  [266] = {x=-22.822, y=-115.715, z=4.852, rx=175.392, ry=-0.809, rz=115, fatherId=fPrdFrame[0]}
  [267] = {x=-24.305, y=-115.715, z=4.874, rx=175.392, ry=-0.869, rz=115, fatherId=fPrdFrame[0]}
  [268] = {x=-25.789, y=-115.715, z=4.897, rx=175.392, ry=-0.928, rz=115, fatherId=fPrdFrame[0]}
  [269] = {x=-27.272, y=-115.714, z=4.922, rx=175.392, ry=-0.987, rz=115, fatherId=fPrdFrame[0]}
  [270] = {x=-28.756, y=-115.714, z=4.949, rx=175.392, ry=-1.046, rz=115, fatherId=fPrdFrame[0]}
  [271] = {x=-30.239, y=-115.714, z=4.977, rx=175.391, ry=-1.105, rz=115, fatherId=fPrdFrame[0]}
  [272] = {x=-31.723, y=-115.714, z=5.007, rx=175.391, ry=-1.165, rz=115, fatherId=fPrdFrame[0]}
  [273] = {x=-33.206, y=-115.714, z=5.038, rx=175.391, ry=-1.224, rz=115, fatherId=fPrdFrame[0]}
  [274] = {x=-34.69, y=-115.714, z=5.071, rx=175.391, ry=-1.283, rz=115, fatherId=fPrdFrame[0]}
  [275] = {x=-36.173, y=-115.714, z=5.105, rx=175.391, ry=-1.342, rz=115, fatherId=fPrdFrame[0]}
  [276] = {x=-37.657, y=-115.714, z=5.141, rx=175.391, ry=-1.401, rz=115, fatherId=fPrdFrame[0]}
  [277] = {x=-39.14, y=-115.714, z=5.179, rx=175.391, ry=-1.461, rz=115, fatherId=fPrdFrame[0]}
  [278] = {x=-40.624, y=-115.714, z=5.218, rx=175.391, ry=-1.52, rz=115, fatherId=fPrdFrame[0]}
  [279] = {x=-42.107, y=-115.714, z=5.258, rx=175.391, ry=-1.579, rz=115, fatherId=fPrdFrame[0]}
  [280] = {x=-43.591, y=-115.714, z=5.301, rx=175.39, ry=-1.638, rz=115, fatherId=fPrdFrame[0]}
  [281] = {x=-45.074, y=-115.714, z=5.344, rx=175.39, ry=-1.698, rz=115, fatherId=fPrdFrame[0]}
  [282] = {x=-46.557, y=-115.714, z=5.389, rx=175.39, ry=-1.757, rz=115, fatherId=fPrdFrame[0]}
  [283] = {x=-48.041, y=-115.714, z=5.436, rx=175.39, ry=-1.816, rz=115, fatherId=fPrdFrame[0]}
  [284] = {x=-49.524, y=-115.714, z=5.485, rx=175.39, ry=-1.875, rz=115, fatherId=fPrdFrame[0]}
  [285] = {x=-52.491, y=-114.23, z=5.466, rx=175.449, ry=-1.994, rz=115, fatherId=fPrdFrame[0]}
  [286] = {x=-51.008, y=-114.23, z=5.414, rx=175.449, ry=-1.934, rz=115, fatherId=fPrdFrame[0]}
  [287] = {x=-49.524, y=-114.23, z=5.364, rx=175.449, ry=-1.875, rz=115, fatherId=fPrdFrame[0]}
  [288] = {x=-48.041, y=-114.231, z=5.316, rx=175.449, ry=-1.816, rz=115, fatherId=fPrdFrame[0]}
  [289] = {x=-46.558, y=-114.231, z=5.269, rx=175.449, ry=-1.757, rz=115, fatherId=fPrdFrame[0]}
  [290] = {x=-45.074, y=-114.231, z=5.224, rx=175.45, ry=-1.697, rz=115, fatherId=fPrdFrame[0]}
  [291] = {x=-43.591, y=-114.231, z=5.18, rx=175.45, ry=-1.638, rz=115, fatherId=fPrdFrame[0]}
  [292] = {x=-42.107, y=-114.231, z=5.138, rx=175.45, ry=-1.579, rz=115, fatherId=fPrdFrame[0]}
  [293] = {x=-40.624, y=-114.231, z=5.098, rx=175.45, ry=-1.52, rz=115, fatherId=fPrdFrame[0]}
  [294] = {x=-39.14, y=-114.231, z=5.059, rx=175.45, ry=-1.461, rz=115, fatherId=fPrdFrame[0]}
  [295] = {x=-37.657, y=-114.231, z=5.021, rx=175.45, ry=-1.401, rz=115, fatherId=fPrdFrame[0]}
  [296] = {x=-36.173, y=-114.231, z=4.985, rx=175.45, ry=-1.342, rz=115, fatherId=fPrdFrame[0]}
  [297] = {x=-34.69, y=-114.231, z=4.951, rx=175.45, ry=-1.283, rz=115, fatherId=fPrdFrame[0]}
  [298] = {x=-33.206, y=-114.231, z=4.918, rx=175.45, ry=-1.224, rz=115, fatherId=fPrdFrame[0]}
  [299] = {x=-31.723, y=-114.231, z=4.887, rx=175.451, ry=-1.164, rz=115, fatherId=fPrdFrame[0]}
  [300] = {x=-30.239, y=-114.231, z=4.857, rx=175.451, ry=-1.105, rz=115, fatherId=fPrdFrame[0]}
  [301] = {x=-28.756, y=-114.231, z=4.829, rx=175.451, ry=-1.046, rz=115, fatherId=fPrdFrame[0]}
  [302] = {x=-27.272, y=-114.231, z=4.802, rx=175.451, ry=-0.987, rz=115, fatherId=fPrdFrame[0]}
  [303] = {x=-25.789, y=-114.231, z=4.777, rx=175.451, ry=-0.928, rz=115, fatherId=fPrdFrame[0]}
  [304] = {x=-24.305, y=-114.231, z=4.754, rx=175.451, ry=-0.868, rz=115, fatherId=fPrdFrame[0]}
  [305] = {x=-22.822, y=-114.231, z=4.732, rx=175.451, ry=-0.809, rz=115, fatherId=fPrdFrame[0]}
  [306] = {x=-21.339, y=-114.231, z=4.711, rx=175.451, ry=-0.75, rz=115, fatherId=fPrdFrame[0]}
  [307] = {x=-19.855, y=-114.231, z=4.693, rx=175.451, ry=-0.691, rz=115, fatherId=fPrdFrame[0]}
  [308] = {x=-18.372, y=-114.231, z=4.675, rx=175.451, ry=-0.632, rz=115, fatherId=fPrdFrame[0]}
  [309] = {x=-16.888, y=-114.231, z=4.659, rx=175.451, ry=-0.572, rz=115, fatherId=fPrdFrame[0]}
  [310] = {x=-15.405, y=-114.231, z=4.645, rx=175.451, ry=-0.513, rz=115, fatherId=fPrdFrame[0]}
  [311] = {x=-13.921, y=-114.231, z=4.633, rx=175.451, ry=-0.454, rz=115, fatherId=fPrdFrame[0]}
  [312] = {x=-12.438, y=-114.231, z=4.621, rx=175.451, ry=-0.395, rz=115, fatherId=fPrdFrame[0]}
  [313] = {x=-10.954, y=-114.231, z=4.612, rx=175.451, ry=-0.336, rz=115, fatherId=fPrdFrame[0]}
  [314] = {x=-9.471, y=-114.231, z=4.604, rx=175.451, ry=-0.276, rz=115, fatherId=fPrdFrame[0]}
  [315] = {x=-7.987, y=-114.231, z=4.597, rx=175.451, ry=-0.217, rz=115, fatherId=fPrdFrame[0]}
  [316] = {x=-6.504, y=-114.231, z=4.592, rx=175.451, ry=-0.158, rz=115, fatherId=fPrdFrame[0]}
  [317] = {x=-5.02, y=-114.231, z=4.589, rx=175.451, ry=-0.099, rz=115, fatherId=fPrdFrame[0]}
  [318] = {x=-3.537, y=-114.231, z=4.587, rx=175.451, ry=-0.04, rz=115, fatherId=fPrdFrame[0]}
  [319] = {x=-2.053, y=-114.231, z=4.587, rx=175.451, ry=0.02, rz=115, fatherId=fPrdFrame[0]}
  [320] = {x=-0.57, y=-114.231, z=4.588, rx=175.451, ry=0.079, rz=115, fatherId=fPrdFrame[0]}
  [321] = {x=0.913, y=-114.231, z=4.591, rx=175.451, ry=0.138, rz=115, fatherId=fPrdFrame[0]}
  [322] = {x=2.397, y=-114.231, z=4.596, rx=175.451, ry=0.197, rz=115, fatherId=fPrdFrame[0]}
  [323] = {x=3.88, y=-114.231, z=4.601, rx=175.451, ry=0.256, rz=115, fatherId=fPrdFrame[0]}
  [324] = {x=5.364, y=-114.231, z=4.609, rx=175.451, ry=0.316, rz=115, fatherId=fPrdFrame[0]}
  [325] = {x=6.847, y=-114.231, z=4.618, rx=175.451, ry=0.375, rz=115, fatherId=fPrdFrame[0]}
  [326] = {x=8.331, y=-114.231, z=4.629, rx=175.451, ry=0.434, rz=115, fatherId=fPrdFrame[0]}
  [327] = {x=9.814, y=-114.231, z=4.641, rx=175.451, ry=0.493, rz=115, fatherId=fPrdFrame[0]}
  [328] = {x=11.298, y=-114.231, z=4.654, rx=175.451, ry=0.552, rz=115, fatherId=fPrdFrame[0]}
  [329] = {x=12.781, y=-114.231, z=4.67, rx=175.451, ry=0.612, rz=115, fatherId=fPrdFrame[0]}
  [330] = {x=14.265, y=-114.231, z=4.686, rx=175.451, ry=0.671, rz=115, fatherId=fPrdFrame[0]}
  [331] = {x=15.748, y=-114.231, z=4.705, rx=175.451, ry=0.73, rz=115, fatherId=fPrdFrame[0]}
  [332] = {x=17.232, y=-114.231, z=4.725, rx=175.451, ry=0.789, rz=115, fatherId=fPrdFrame[0]}
  [333] = {x=18.715, y=-114.231, z=4.746, rx=175.451, ry=0.848, rz=115, fatherId=fPrdFrame[0]}
  [334] = {x=20.199, y=-114.231, z=4.769, rx=175.451, ry=0.908, rz=115, fatherId=fPrdFrame[0]}
  [335] = {x=21.682, y=-114.231, z=4.794, rx=175.451, ry=0.967, rz=115, fatherId=fPrdFrame[0]}
  [336] = {x=23.166, y=-114.231, z=4.82, rx=175.451, ry=1.026, rz=115, fatherId=fPrdFrame[0]}
  [337] = {x=24.649, y=-114.231, z=4.847, rx=175.451, ry=1.085, rz=115, fatherId=fPrdFrame[0]}
  [338] = {x=26.132, y=-114.231, z=4.877, rx=175.451, ry=1.144, rz=115, fatherId=fPrdFrame[0]}
  [339] = {x=27.616, y=-114.231, z=4.907, rx=175.45, ry=1.204, rz=115, fatherId=fPrdFrame[0]}
  [340] = {x=29.099, y=-114.231, z=4.94, rx=175.45, ry=1.263, rz=115, fatherId=fPrdFrame[0]}
  [341] = {x=30.583, y=-114.231, z=4.973, rx=175.45, ry=1.322, rz=115, fatherId=fPrdFrame[0]}
  [342] = {x=32.066, y=-114.231, z=5.009, rx=175.45, ry=1.381, rz=115, fatherId=fPrdFrame[0]}
  [343] = {x=33.55, y=-114.231, z=5.046, rx=175.45, ry=1.44, rz=115, fatherId=fPrdFrame[0]}
  [344] = {x=35.033, y=-114.231, z=5.084, rx=175.45, ry=1.5, rz=115, fatherId=fPrdFrame[0]}
  [345] = {x=36.517, y=-114.231, z=5.124, rx=175.45, ry=1.559, rz=115, fatherId=fPrdFrame[0]}
  [346] = {x=38, y=-114.231, z=5.166, rx=175.45, ry=1.618, rz=115, fatherId=fPrdFrame[0]}
  [347] = {x=39.484, y=-114.231, z=5.209, rx=175.45, ry=1.677, rz=115, fatherId=fPrdFrame[0]}
  [348] = {x=40.967, y=-114.231, z=5.254, rx=175.449, ry=1.736, rz=115, fatherId=fPrdFrame[0]}
  [349] = {x=42.451, y=-114.231, z=5.3, rx=175.449, ry=1.796, rz=115, fatherId=fPrdFrame[0]}
  [350] = {x=43.934, y=-114.23, z=5.348, rx=175.449, ry=1.855, rz=115, fatherId=fPrdFrame[0]}
  [351] = {x=45.418, y=-114.23, z=5.397, rx=175.449, ry=1.914, rz=115, fatherId=fPrdFrame[0]}
  [352] = {x=46.901, y=-114.23, z=5.448, rx=175.449, ry=1.973, rz=115, fatherId=fPrdFrame[0]}
  [353] = {x=51.351, y=-112.747, z=5.491, rx=175.508, ry=2.151, rz=115, fatherId=fPrdFrame[0]}
  [354] = {x=49.868, y=-112.747, z=5.436, rx=175.508, ry=2.092, rz=115, fatherId=fPrdFrame[0]}
  [355] = {x=48.385, y=-112.747, z=5.382, rx=175.508, ry=2.032, rz=115, fatherId=fPrdFrame[0]}
  [356] = {x=46.901, y=-112.747, z=5.329, rx=175.508, ry=1.973, rz=115, fatherId=fPrdFrame[0]}
  [357] = {x=45.418, y=-112.747, z=5.278, rx=175.508, ry=1.914, rz=115, fatherId=fPrdFrame[0]}
  [358] = {x=43.934, y=-112.747, z=5.229, rx=175.508, ry=1.855, rz=115, fatherId=fPrdFrame[0]}
  [359] = {x=42.451, y=-112.747, z=5.181, rx=175.508, ry=1.796, rz=115, fatherId=fPrdFrame[0]}
  [360] = {x=40.967, y=-112.747, z=5.135, rx=175.509, ry=1.736, rz=115, fatherId=fPrdFrame[0]}
  [361] = {x=39.484, y=-112.747, z=5.09, rx=175.509, ry=1.677, rz=115, fatherId=fPrdFrame[0]}
  [362] = {x=38, y=-112.747, z=5.047, rx=175.509, ry=1.618, rz=115, fatherId=fPrdFrame[0]}
  [363] = {x=36.517, y=-112.747, z=5.006, rx=175.509, ry=1.559, rz=115, fatherId=fPrdFrame[0]}
  [364] = {x=35.033, y=-112.747, z=4.966, rx=175.509, ry=1.499, rz=115, fatherId=fPrdFrame[0]}
  [365] = {x=33.55, y=-112.747, z=4.927, rx=175.509, ry=1.44, rz=115, fatherId=fPrdFrame[0]}
  [366] = {x=32.066, y=-112.747, z=4.89, rx=175.509, ry=1.381, rz=115, fatherId=fPrdFrame[0]}
  [367] = {x=30.583, y=-112.747, z=4.855, rx=175.51, ry=1.322, rz=115, fatherId=fPrdFrame[0]}
  [368] = {x=29.099, y=-112.747, z=4.821, rx=175.51, ry=1.263, rz=115, fatherId=fPrdFrame[0]}
  [369] = {x=27.616, y=-112.747, z=4.789, rx=175.51, ry=1.203, rz=115, fatherId=fPrdFrame[0]}
  [370] = {x=26.132, y=-112.747, z=4.758, rx=175.51, ry=1.144, rz=115, fatherId=fPrdFrame[0]}
  [371] = {x=24.649, y=-112.747, z=4.729, rx=175.51, ry=1.085, rz=115, fatherId=fPrdFrame[0]}
  [372] = {x=23.166, y=-112.747, z=4.701, rx=175.51, ry=1.026, rz=115, fatherId=fPrdFrame[0]}
  [373] = {x=21.682, y=-112.747, z=4.675, rx=175.51, ry=0.967, rz=115, fatherId=fPrdFrame[0]}
  [374] = {x=20.199, y=-112.747, z=4.651, rx=175.51, ry=0.907, rz=115, fatherId=fPrdFrame[0]}
  [375] = {x=18.715, y=-112.747, z=4.628, rx=175.51, ry=0.848, rz=115, fatherId=fPrdFrame[0]}
  [376] = {x=17.232, y=-112.748, z=4.606, rx=175.51, ry=0.789, rz=115, fatherId=fPrdFrame[0]}
  [377] = {x=15.748, y=-112.748, z=4.586, rx=175.51, ry=0.73, rz=115, fatherId=fPrdFrame[0]}
  [378] = {x=14.265, y=-112.748, z=4.568, rx=175.51, ry=0.671, rz=115, fatherId=fPrdFrame[0]}
  [379] = {x=12.781, y=-112.748, z=4.551, rx=175.51, ry=0.611, rz=115, fatherId=fPrdFrame[0]}
  [380] = {x=11.298, y=-112.748, z=4.536, rx=175.51, ry=0.552, rz=115, fatherId=fPrdFrame[0]}
  [381] = {x=9.814, y=-112.748, z=4.522, rx=175.511, ry=0.493, rz=115, fatherId=fPrdFrame[0]}
  [382] = {x=8.331, y=-112.748, z=4.51, rx=175.511, ry=0.434, rz=115, fatherId=fPrdFrame[0]}
  [383] = {x=6.847, y=-112.748, z=4.499, rx=175.511, ry=0.375, rz=115, fatherId=fPrdFrame[0]}
  [384] = {x=5.364, y=-112.748, z=4.49, rx=175.511, ry=0.315, rz=115, fatherId=fPrdFrame[0]}
  [385] = {x=3.88, y=-112.748, z=4.483, rx=175.511, ry=0.256, rz=115, fatherId=fPrdFrame[0]}
  [386] = {x=2.397, y=-112.748, z=4.477, rx=175.511, ry=0.197, rz=115, fatherId=fPrdFrame[0]}
  [387] = {x=0.913, y=-112.748, z=4.473, rx=175.511, ry=0.138, rz=115, fatherId=fPrdFrame[0]}
  [388] = {x=-0.57, y=-112.748, z=4.47, rx=175.511, ry=0.079, rz=115, fatherId=fPrdFrame[0]}
  [389] = {x=-2.053, y=-112.748, z=4.469, rx=175.511, ry=0.02, rz=115, fatherId=fPrdFrame[0]}
  [390] = {x=-3.537, y=-112.748, z=4.469, rx=175.511, ry=-0.04, rz=115, fatherId=fPrdFrame[0]}
  [391] = {x=-5.02, y=-112.748, z=4.471, rx=175.511, ry=-0.099, rz=115, fatherId=fPrdFrame[0]}
  [392] = {x=-6.504, y=-112.748, z=4.474, rx=175.511, ry=-0.158, rz=115, fatherId=fPrdFrame[0]}
  [393] = {x=-7.987, y=-112.748, z=4.479, rx=175.511, ry=-0.217, rz=115, fatherId=fPrdFrame[0]}
  [394] = {x=-9.471, y=-112.748, z=4.485, rx=175.511, ry=-0.276, rz=115, fatherId=fPrdFrame[0]}
  [395] = {x=-10.954, y=-112.748, z=4.493, rx=175.511, ry=-0.336, rz=115, fatherId=fPrdFrame[0]}
  [396] = {x=-12.438, y=-112.748, z=4.503, rx=175.511, ry=-0.395, rz=115, fatherId=fPrdFrame[0]}
  [397] = {x=-13.921, y=-112.748, z=4.514, rx=175.511, ry=-0.454, rz=115, fatherId=fPrdFrame[0]}
  [398] = {x=-15.405, y=-112.748, z=4.527, rx=175.511, ry=-0.513, rz=115, fatherId=fPrdFrame[0]}
  [399] = {x=-16.888, y=-112.748, z=4.541, rx=175.51, ry=-0.572, rz=115, fatherId=fPrdFrame[0]}
  [400] = {x=-18.372, y=-112.748, z=4.557, rx=175.51, ry=-0.632, rz=115, fatherId=fPrdFrame[0]}
  [401] = {x=-19.855, y=-112.748, z=4.574, rx=175.51, ry=-0.691, rz=115, fatherId=fPrdFrame[0]}
  [402] = {x=-21.339, y=-112.748, z=4.593, rx=175.51, ry=-0.75, rz=115, fatherId=fPrdFrame[0]}
  [403] = {x=-22.822, y=-112.748, z=4.613, rx=175.51, ry=-0.809, rz=115, fatherId=fPrdFrame[0]}
  [404] = {x=-24.306, y=-112.747, z=4.635, rx=175.51, ry=-0.868, rz=115, fatherId=fPrdFrame[0]}
  [405] = {x=-25.789, y=-112.747, z=4.659, rx=175.51, ry=-0.928, rz=115, fatherId=fPrdFrame[0]}
  [406] = {x=-27.272, y=-112.747, z=4.684, rx=175.51, ry=-0.987, rz=115, fatherId=fPrdFrame[0]}
  [407] = {x=-28.756, y=-112.747, z=4.71, rx=175.51, ry=-1.046, rz=115, fatherId=fPrdFrame[0]}
  [408] = {x=-30.239, y=-112.747, z=4.739, rx=175.51, ry=-1.105, rz=115, fatherId=fPrdFrame[0]}
  [409] = {x=-31.723, y=-112.747, z=4.768, rx=175.51, ry=-1.164, rz=115, fatherId=fPrdFrame[0]}
  [410] = {x=-33.206, y=-112.747, z=4.799, rx=175.51, ry=-1.224, rz=115, fatherId=fPrdFrame[0]}
  [411] = {x=-34.69, y=-112.747, z=4.832, rx=175.51, ry=-1.283, rz=115, fatherId=fPrdFrame[0]}
  [412] = {x=-36.173, y=-112.747, z=4.867, rx=175.509, ry=-1.342, rz=115, fatherId=fPrdFrame[0]}
  [413] = {x=-37.657, y=-112.747, z=4.903, rx=175.509, ry=-1.401, rz=115, fatherId=fPrdFrame[0]}
  [414] = {x=-39.14, y=-112.747, z=4.94, rx=175.509, ry=-1.46, rz=115, fatherId=fPrdFrame[0]}
  [415] = {x=-40.624, y=-112.747, z=4.979, rx=175.509, ry=-1.52, rz=115, fatherId=fPrdFrame[0]}
  [416] = {x=-42.107, y=-112.747, z=5.02, rx=175.509, ry=-1.579, rz=115, fatherId=fPrdFrame[0]}
  [417] = {x=-43.591, y=-112.747, z=5.062, rx=175.509, ry=-1.638, rz=115, fatherId=fPrdFrame[0]}
  [418] = {x=-45.074, y=-112.747, z=5.105, rx=175.509, ry=-1.697, rz=115, fatherId=fPrdFrame[0]}
  [419] = {x=-46.558, y=-112.747, z=5.151, rx=175.509, ry=-1.756, rz=115, fatherId=fPrdFrame[0]}
  [420] = {x=-48.041, y=-112.747, z=5.197, rx=175.508, ry=-1.816, rz=115, fatherId=fPrdFrame[0]}
  [421] = {x=-49.525, y=-112.747, z=5.246, rx=175.508, ry=-1.875, rz=115, fatherId=fPrdFrame[0]}
  [422] = {x=-51.008, y=-112.747, z=5.296, rx=175.508, ry=-1.934, rz=115, fatherId=fPrdFrame[0]}
  [423] = {x=-52.491, y=-112.747, z=5.347, rx=175.508, ry=-1.993, rz=115, fatherId=fPrdFrame[0]}
  [424] = {x=-53.975, y=-112.747, z=5.4, rx=175.508, ry=-2.053, rz=115, fatherId=fPrdFrame[0]}
  [425] = {x=-55.458, y=-112.747, z=5.455, rx=175.508, ry=-2.112, rz=115, fatherId=fPrdFrame[0]}
  [426] = {x=-58.425, y=-111.263, z=5.451, rx=175.567, ry=-2.23, rz=115, fatherId=fPrdFrame[0]}
  [427] = {x=-56.942, y=-111.263, z=5.394, rx=175.567, ry=-2.171, rz=115, fatherId=fPrdFrame[0]}
  [428] = {x=-55.458, y=-111.263, z=5.338, rx=175.567, ry=-2.112, rz=115, fatherId=fPrdFrame[0]}
  [429] = {x=-53.975, y=-111.263, z=5.283, rx=175.567, ry=-2.052, rz=115, fatherId=fPrdFrame[0]}
  [430] = {x=-52.492, y=-111.263, z=5.23, rx=175.567, ry=-1.993, rz=115, fatherId=fPrdFrame[0]}
  [431] = {x=-51.008, y=-111.263, z=5.179, rx=175.567, ry=-1.934, rz=115, fatherId=fPrdFrame[0]}
  [432] = {x=-49.525, y=-111.263, z=5.129, rx=175.568, ry=-1.875, rz=115, fatherId=fPrdFrame[0]}
  [433] = {x=-48.041, y=-111.263, z=5.08, rx=175.568, ry=-1.816, rz=115, fatherId=fPrdFrame[0]}
  [434] = {x=-46.558, y=-111.264, z=5.034, rx=175.568, ry=-1.756, rz=115, fatherId=fPrdFrame[0]}
  [435] = {x=-45.074, y=-111.264, z=4.988, rx=175.568, ry=-1.697, rz=115, fatherId=fPrdFrame[0]}
  [436] = {x=-43.591, y=-111.264, z=4.945, rx=175.568, ry=-1.638, rz=115, fatherId=fPrdFrame[0]}
  [437] = {x=-42.107, y=-111.264, z=4.903, rx=175.568, ry=-1.579, rz=115, fatherId=fPrdFrame[0]}
  [438] = {x=-40.624, y=-111.264, z=4.862, rx=175.568, ry=-1.519, rz=115, fatherId=fPrdFrame[0]}
  [439] = {x=-39.14, y=-111.264, z=4.823, rx=175.568, ry=-1.46, rz=115, fatherId=fPrdFrame[0]}
  [440] = {x=-37.657, y=-111.264, z=4.786, rx=175.569, ry=-1.401, rz=115, fatherId=fPrdFrame[0]}
  [441] = {x=-36.173, y=-111.264, z=4.75, rx=175.569, ry=-1.342, rz=115, fatherId=fPrdFrame[0]}
  [442] = {x=-34.69, y=-111.264, z=4.715, rx=175.569, ry=-1.283, rz=115, fatherId=fPrdFrame[0]}
  [443] = {x=-33.206, y=-111.264, z=4.682, rx=175.569, ry=-1.223, rz=115, fatherId=fPrdFrame[0]}
  [444] = {x=-31.723, y=-111.264, z=4.651, rx=175.569, ry=-1.164, rz=115, fatherId=fPrdFrame[0]}
  [445] = {x=-30.239, y=-111.264, z=4.622, rx=175.569, ry=-1.105, rz=115, fatherId=fPrdFrame[0]}
  [446] = {x=-28.756, y=-111.264, z=4.593, rx=175.569, ry=-1.046, rz=115, fatherId=fPrdFrame[0]}
  [447] = {x=-27.272, y=-111.264, z=4.567, rx=175.569, ry=-0.987, rz=115, fatherId=fPrdFrame[0]}
  [448] = {x=-25.789, y=-111.264, z=4.542, rx=175.569, ry=-0.927, rz=115, fatherId=fPrdFrame[0]}
  [449] = {x=-24.306, y=-111.264, z=4.518, rx=175.569, ry=-0.868, rz=115, fatherId=fPrdFrame[0]}
  [450] = {x=-22.822, y=-111.264, z=4.496, rx=175.569, ry=-0.809, rz=115, fatherId=fPrdFrame[0]}
  [451] = {x=-21.339, y=-111.264, z=4.476, rx=175.57, ry=-0.75, rz=115, fatherId=fPrdFrame[0]}
  [452] = {x=-19.855, y=-111.264, z=4.457, rx=175.57, ry=-0.691, rz=115, fatherId=fPrdFrame[0]}
  [453] = {x=-18.372, y=-111.264, z=4.44, rx=175.57, ry=-0.632, rz=115, fatherId=fPrdFrame[0]}
  [454] = {x=-16.888, y=-111.264, z=4.424, rx=175.57, ry=-0.572, rz=115, fatherId=fPrdFrame[0]}
  [455] = {x=-15.405, y=-111.264, z=4.41, rx=175.57, ry=-0.513, rz=115, fatherId=fPrdFrame[0]}
  [456] = {x=-13.921, y=-111.264, z=4.397, rx=175.57, ry=-0.454, rz=115, fatherId=fPrdFrame[0]}
  [457] = {x=-12.438, y=-111.264, z=4.386, rx=175.57, ry=-0.395, rz=115, fatherId=fPrdFrame[0]}
  [458] = {x=-10.954, y=-111.264, z=4.376, rx=175.57, ry=-0.336, rz=115, fatherId=fPrdFrame[0]}
  [459] = {x=-9.471, y=-111.264, z=4.368, rx=175.57, ry=-0.276, rz=115, fatherId=fPrdFrame[0]}
  [460] = {x=-7.987, y=-111.264, z=4.362, rx=175.57, ry=-0.217, rz=115, fatherId=fPrdFrame[0]}
  [461] = {x=-6.504, y=-111.264, z=4.357, rx=175.57, ry=-0.158, rz=115, fatherId=fPrdFrame[0]}
  [462] = {x=-5.02, y=-111.264, z=4.354, rx=175.57, ry=-0.099, rz=115, fatherId=fPrdFrame[0]}
  [463] = {x=-3.537, y=-111.264, z=4.352, rx=175.57, ry=-0.04, rz=115, fatherId=fPrdFrame[0]}
  [464] = {x=-2.053, y=-111.264, z=4.352, rx=175.57, ry=0.02, rz=115, fatherId=fPrdFrame[0]}
  [465] = {x=-0.57, y=-111.264, z=4.353, rx=175.57, ry=0.079, rz=115, fatherId=fPrdFrame[0]}
  [466] = {x=0.913, y=-111.264, z=4.356, rx=175.57, ry=0.138, rz=115, fatherId=fPrdFrame[0]}
  [467] = {x=2.397, y=-111.264, z=4.36, rx=175.57, ry=0.197, rz=115, fatherId=fPrdFrame[0]}
  [468] = {x=3.88, y=-111.264, z=4.366, rx=175.57, ry=0.256, rz=115, fatherId=fPrdFrame[0]}
  [469] = {x=5.364, y=-111.264, z=4.373, rx=175.57, ry=0.315, rz=115, fatherId=fPrdFrame[0]}
  [470] = {x=6.847, y=-111.264, z=4.382, rx=175.57, ry=0.375, rz=115, fatherId=fPrdFrame[0]}
  [471] = {x=8.331, y=-111.264, z=4.393, rx=175.57, ry=0.434, rz=115, fatherId=fPrdFrame[0]}
  [472] = {x=9.814, y=-111.264, z=4.405, rx=175.57, ry=0.493, rz=115, fatherId=fPrdFrame[0]}
  [473] = {x=11.298, y=-111.264, z=4.419, rx=175.57, ry=0.552, rz=115, fatherId=fPrdFrame[0]}
  [474] = {x=12.781, y=-111.264, z=4.434, rx=175.57, ry=0.611, rz=115, fatherId=fPrdFrame[0]}
  [475] = {x=14.265, y=-111.264, z=4.451, rx=175.57, ry=0.671, rz=115, fatherId=fPrdFrame[0]}
  [476] = {x=15.748, y=-111.264, z=4.469, rx=175.57, ry=0.73, rz=115, fatherId=fPrdFrame[0]}
  [477] = {x=17.232, y=-111.264, z=4.489, rx=175.569, ry=0.789, rz=115, fatherId=fPrdFrame[0]}
  [478] = {x=18.715, y=-111.264, z=4.511, rx=175.569, ry=0.848, rz=115, fatherId=fPrdFrame[0]}
  [479] = {x=20.199, y=-111.264, z=4.534, rx=175.569, ry=0.907, rz=115, fatherId=fPrdFrame[0]}
  [480] = {x=21.682, y=-111.264, z=4.558, rx=175.569, ry=0.967, rz=115, fatherId=fPrdFrame[0]}
  [481] = {x=23.166, y=-111.264, z=4.584, rx=175.569, ry=1.026, rz=115, fatherId=fPrdFrame[0]}
  [482] = {x=24.649, y=-111.264, z=4.612, rx=175.569, ry=1.085, rz=115, fatherId=fPrdFrame[0]}
  [483] = {x=26.133, y=-111.264, z=4.641, rx=175.569, ry=1.144, rz=115, fatherId=fPrdFrame[0]}
  [484] = {x=27.616, y=-111.264, z=4.672, rx=175.569, ry=1.203, rz=115, fatherId=fPrdFrame[0]}
  [485] = {x=29.099, y=-111.264, z=4.704, rx=175.569, ry=1.263, rz=115, fatherId=fPrdFrame[0]}
  [486] = {x=30.583, y=-111.264, z=4.738, rx=175.569, ry=1.322, rz=115, fatherId=fPrdFrame[0]}
  [487] = {x=32.066, y=-111.264, z=4.773, rx=175.569, ry=1.381, rz=115, fatherId=fPrdFrame[0]}
  [488] = {x=33.55, y=-111.264, z=4.81, rx=175.568, ry=1.44, rz=115, fatherId=fPrdFrame[0]}
  [489] = {x=35.033, y=-111.264, z=4.849, rx=175.568, ry=1.499, rz=115, fatherId=fPrdFrame[0]}
  [490] = {x=36.517, y=-111.264, z=4.889, rx=175.568, ry=1.559, rz=115, fatherId=fPrdFrame[0]}
  [491] = {x=38, y=-111.264, z=4.93, rx=175.568, ry=1.618, rz=115, fatherId=fPrdFrame[0]}
  [492] = {x=39.484, y=-111.264, z=4.973, rx=175.568, ry=1.677, rz=115, fatherId=fPrdFrame[0]}
  [493] = {x=40.967, y=-111.264, z=5.018, rx=175.568, ry=1.736, rz=115, fatherId=fPrdFrame[0]}
  [494] = {x=42.451, y=-111.264, z=5.064, rx=175.568, ry=1.795, rz=115, fatherId=fPrdFrame[0]}
  [495] = {x=43.934, y=-111.263, z=5.112, rx=175.568, ry=1.855, rz=115, fatherId=fPrdFrame[0]}
  [496] = {x=45.418, y=-111.263, z=5.161, rx=175.567, ry=1.914, rz=115, fatherId=fPrdFrame[0]}
  [497] = {x=46.901, y=-111.263, z=5.212, rx=175.567, ry=1.973, rz=115, fatherId=fPrdFrame[0]}
  [498] = {x=48.385, y=-111.263, z=5.265, rx=175.567, ry=2.032, rz=115, fatherId=fPrdFrame[0]}
  [499] = {x=49.868, y=-111.263, z=5.319, rx=175.567, ry=2.092, rz=115, fatherId=fPrdFrame[0]}
  [500] = {x=51.352, y=-111.263, z=5.374, rx=175.567, ry=2.151, rz=115, fatherId=fPrdFrame[0]}
  [501] = {x=52.835, y=-111.263, z=5.431, rx=175.567, ry=2.21, rz=115, fatherId=fPrdFrame[0]}
  [502] = {x=54.318, y=-111.263, z=5.49, rx=175.566, ry=2.269, rz=115, fatherId=fPrdFrame[0]}
  [503] = {x=57.285, y=-109.78, z=5.497, rx=175.625, ry=2.387, rz=115, fatherId=fPrdFrame[0]}
  [504] = {x=55.802, y=-109.78, z=5.435, rx=175.625, ry=2.328, rz=115, fatherId=fPrdFrame[0]}
  [505] = {x=54.319, y=-109.78, z=5.375, rx=175.626, ry=2.269, rz=115, fatherId=fPrdFrame[0]}
  [506] = {x=52.835, y=-109.78, z=5.316, rx=175.626, ry=2.21, rz=115, fatherId=fPrdFrame[0]}
  [507] = {x=51.352, y=-109.78, z=5.259, rx=175.626, ry=2.151, rz=115, fatherId=fPrdFrame[0]}
  [508] = {x=49.868, y=-109.78, z=5.203, rx=175.626, ry=2.091, rz=115, fatherId=fPrdFrame[0]}
  [509] = {x=48.385, y=-109.78, z=5.149, rx=175.626, ry=2.032, rz=115, fatherId=fPrdFrame[0]}
  [510] = {x=46.901, y=-109.78, z=5.097, rx=175.626, ry=1.973, rz=115, fatherId=fPrdFrame[0]}
  [511] = {x=45.418, y=-109.78, z=5.046, rx=175.627, ry=1.914, rz=115, fatherId=fPrdFrame[0]}
  [512] = {x=43.934, y=-109.78, z=4.997, rx=175.627, ry=1.854, rz=115, fatherId=fPrdFrame[0]}
  [513] = {x=42.451, y=-109.78, z=4.949, rx=175.627, ry=1.795, rz=115, fatherId=fPrdFrame[0]}
  [514] = {x=40.967, y=-109.78, z=4.903, rx=175.627, ry=1.736, rz=115, fatherId=fPrdFrame[0]}
  [515] = {x=39.484, y=-109.78, z=4.858, rx=175.627, ry=1.677, rz=115, fatherId=fPrdFrame[0]}
  [516] = {x=38, y=-109.78, z=4.815, rx=175.627, ry=1.618, rz=115, fatherId=fPrdFrame[0]}
  [517] = {x=36.517, y=-109.78, z=4.773, rx=175.627, ry=1.558, rz=115, fatherId=fPrdFrame[0]}
  [518] = {x=35.033, y=-109.78, z=4.733, rx=175.628, ry=1.499, rz=115, fatherId=fPrdFrame[0]}
  [519] = {x=33.55, y=-109.78, z=4.695, rx=175.628, ry=1.44, rz=115, fatherId=fPrdFrame[0]}
  [520] = {x=32.066, y=-109.78, z=4.658, rx=175.628, ry=1.381, rz=115, fatherId=fPrdFrame[0]}
  [521] = {x=30.583, y=-109.78, z=4.622, rx=175.628, ry=1.322, rz=115, fatherId=fPrdFrame[0]}
  [522] = {x=29.099, y=-109.78, z=4.588, rx=175.628, ry=1.262, rz=115, fatherId=fPrdFrame[0]}
  [523] = {x=27.616, y=-109.78, z=4.556, rx=175.628, ry=1.203, rz=115, fatherId=fPrdFrame[0]}
  [524] = {x=26.133, y=-109.78, z=4.525, rx=175.628, ry=1.144, rz=115, fatherId=fPrdFrame[0]}
  [525] = {x=24.649, y=-109.78, z=4.496, rx=175.628, ry=1.085, rz=115, fatherId=fPrdFrame[0]}
  [526] = {x=23.166, y=-109.78, z=4.469, rx=175.628, ry=1.026, rz=115, fatherId=fPrdFrame[0]}
  [527] = {x=21.682, y=-109.78, z=4.443, rx=175.628, ry=0.966, rz=115, fatherId=fPrdFrame[0]}
  [528] = {x=20.199, y=-109.78, z=4.418, rx=175.629, ry=0.907, rz=115, fatherId=fPrdFrame[0]}
  [529] = {x=18.715, y=-109.78, z=4.395, rx=175.629, ry=0.848, rz=115, fatherId=fPrdFrame[0]}
  [530] = {x=17.232, y=-109.78, z=4.374, rx=175.629, ry=0.789, rz=115, fatherId=fPrdFrame[0]}
  [531] = {x=15.748, y=-109.78, z=4.354, rx=175.629, ry=0.73, rz=115, fatherId=fPrdFrame[0]}
  [532] = {x=14.265, y=-109.781, z=4.335, rx=175.629, ry=0.671, rz=115, fatherId=fPrdFrame[0]}
  [533] = {x=12.781, y=-109.781, z=4.319, rx=175.629, ry=0.611, rz=115, fatherId=fPrdFrame[0]}
  [534] = {x=11.298, y=-109.781, z=4.303, rx=175.629, ry=0.552, rz=115, fatherId=fPrdFrame[0]}
  [535] = {x=9.814, y=-109.781, z=4.29, rx=175.629, ry=0.493, rz=115, fatherId=fPrdFrame[0]}
  [536] = {x=8.331, y=-109.781, z=4.278, rx=175.629, ry=0.434, rz=115, fatherId=fPrdFrame[0]}
  [537] = {x=6.847, y=-109.781, z=4.267, rx=175.629, ry=0.375, rz=115, fatherId=fPrdFrame[0]}
  [538] = {x=5.364, y=-109.781, z=4.258, rx=175.629, ry=0.315, rz=115, fatherId=fPrdFrame[0]}
  [539] = {x=3.88, y=-109.781, z=4.251, rx=175.629, ry=0.256, rz=115, fatherId=fPrdFrame[0]}
  [540] = {x=2.397, y=-109.781, z=4.245, rx=175.629, ry=0.197, rz=115, fatherId=fPrdFrame[0]}
  [541] = {x=0.913, y=-109.781, z=4.24, rx=175.629, ry=0.138, rz=115, fatherId=fPrdFrame[0]}
  [542] = {x=-0.57, y=-109.781, z=4.237, rx=175.629, ry=0.079, rz=115, fatherId=fPrdFrame[0]}
  [543] = {x=-2.053, y=-109.781, z=4.236, rx=175.629, ry=0.02, rz=115, fatherId=fPrdFrame[0]}
  [544] = {x=-3.537, y=-109.781, z=4.236, rx=175.629, ry=-0.04, rz=115, fatherId=fPrdFrame[0]}
  [545] = {x=-5.02, y=-109.781, z=4.238, rx=175.629, ry=-0.099, rz=115, fatherId=fPrdFrame[0]}
  [546] = {x=-6.504, y=-109.781, z=4.242, rx=175.629, ry=-0.158, rz=115, fatherId=fPrdFrame[0]}
  [547] = {x=-7.987, y=-109.781, z=4.246, rx=175.629, ry=-0.217, rz=115, fatherId=fPrdFrame[0]}
  [548] = {x=-9.471, y=-109.781, z=4.253, rx=175.629, ry=-0.276, rz=115, fatherId=fPrdFrame[0]}
  [549] = {x=-10.954, y=-109.781, z=4.261, rx=175.629, ry=-0.336, rz=115, fatherId=fPrdFrame[0]}
  [550] = {x=-12.438, y=-109.781, z=4.27, rx=175.629, ry=-0.395, rz=115, fatherId=fPrdFrame[0]}
  [551] = {x=-13.921, y=-109.781, z=4.282, rx=175.629, ry=-0.454, rz=115, fatherId=fPrdFrame[0]}
  [552] = {x=-15.405, y=-109.781, z=4.294, rx=175.629, ry=-0.513, rz=115, fatherId=fPrdFrame[0]}
  [553] = {x=-16.888, y=-109.781, z=4.308, rx=175.629, ry=-0.572, rz=115, fatherId=fPrdFrame[0]}
  [554] = {x=-18.372, y=-109.781, z=4.324, rx=175.629, ry=-0.631, rz=115, fatherId=fPrdFrame[0]}
  [555] = {x=-19.855, y=-109.781, z=4.342, rx=175.629, ry=-0.691, rz=115, fatherId=fPrdFrame[0]}
  [556] = {x=-21.339, y=-109.78, z=4.36, rx=175.629, ry=-0.75, rz=115, fatherId=fPrdFrame[0]}
  [557] = {x=-22.822, y=-109.78, z=4.381, rx=175.629, ry=-0.809, rz=115, fatherId=fPrdFrame[0]}
  [558] = {x=-24.306, y=-109.78, z=4.403, rx=175.629, ry=-0.868, rz=115, fatherId=fPrdFrame[0]}
  [559] = {x=-25.789, y=-109.78, z=4.426, rx=175.628, ry=-0.927, rz=115, fatherId=fPrdFrame[0]}
  [560] = {x=-27.273, y=-109.78, z=4.451, rx=175.628, ry=-0.987, rz=115, fatherId=fPrdFrame[0]}
  [561] = {x=-28.756, y=-109.78, z=4.478, rx=175.628, ry=-1.046, rz=115, fatherId=fPrdFrame[0]}
  [562] = {x=-30.239, y=-109.78, z=4.506, rx=175.628, ry=-1.105, rz=115, fatherId=fPrdFrame[0]}
  [563] = {x=-31.723, y=-109.78, z=4.536, rx=175.628, ry=-1.164, rz=115, fatherId=fPrdFrame[0]}
  [564] = {x=-33.206, y=-109.78, z=4.567, rx=175.628, ry=-1.223, rz=115, fatherId=fPrdFrame[0]}
  [565] = {x=-34.69, y=-109.78, z=4.6, rx=175.628, ry=-1.283, rz=115, fatherId=fPrdFrame[0]}
  [566] = {x=-36.173, y=-109.78, z=4.634, rx=175.628, ry=-1.342, rz=115, fatherId=fPrdFrame[0]}
  [567] = {x=-37.657, y=-109.78, z=4.67, rx=175.628, ry=-1.401, rz=115, fatherId=fPrdFrame[0]}
  [568] = {x=-39.14, y=-109.78, z=4.708, rx=175.628, ry=-1.46, rz=115, fatherId=fPrdFrame[0]}
  [569] = {x=-40.624, y=-109.78, z=4.747, rx=175.628, ry=-1.519, rz=115, fatherId=fPrdFrame[0]}
  [570] = {x=-42.107, y=-109.78, z=4.787, rx=175.627, ry=-1.579, rz=115, fatherId=fPrdFrame[0]}
  [571] = {x=-43.591, y=-109.78, z=4.829, rx=175.627, ry=-1.638, rz=115, fatherId=fPrdFrame[0]}
  [572] = {x=-45.074, y=-109.78, z=4.873, rx=175.627, ry=-1.697, rz=115, fatherId=fPrdFrame[0]}
  [573] = {x=-46.558, y=-109.78, z=4.918, rx=175.627, ry=-1.756, rz=115, fatherId=fPrdFrame[0]}
  [574] = {x=-48.041, y=-109.78, z=4.965, rx=175.627, ry=-1.815, rz=115, fatherId=fPrdFrame[0]}
  [575] = {x=-49.525, y=-109.78, z=5.013, rx=175.627, ry=-1.875, rz=115, fatherId=fPrdFrame[0]}
  [576] = {x=-51.008, y=-109.78, z=5.063, rx=175.627, ry=-1.934, rz=115, fatherId=fPrdFrame[0]}
  [577] = {x=-52.492, y=-109.78, z=5.114, rx=175.626, ry=-1.993, rz=115, fatherId=fPrdFrame[0]}
  [578] = {x=-53.975, y=-109.78, z=5.167, rx=175.626, ry=-2.052, rz=115, fatherId=fPrdFrame[0]}
  [579] = {x=-55.458, y=-109.78, z=5.222, rx=175.626, ry=-2.111, rz=115, fatherId=fPrdFrame[0]}
  [580] = {x=-56.942, y=-109.78, z=5.278, rx=175.626, ry=-2.171, rz=115, fatherId=fPrdFrame[0]}
  [581] = {x=-58.425, y=-109.78, z=5.336, rx=175.626, ry=-2.23, rz=115, fatherId=fPrdFrame[0]}
  [582] = {x=-59.909, y=-109.78, z=5.395, rx=175.626, ry=-2.289, rz=115, fatherId=fPrdFrame[0]}
  [583] = {x=-61.392, y=-109.78, z=5.456, rx=175.625, ry=-2.348, rz=115, fatherId=fPrdFrame[0]}
  [584] = {x=-64.359, y=-108.296, z=5.468, rx=175.684, ry=-2.467, rz=115, fatherId=fPrdFrame[0]}
  [585] = {x=-62.876, y=-108.296, z=5.404, rx=175.684, ry=-2.407, rz=115, fatherId=fPrdFrame[0]}
  [586] = {x=-61.392, y=-108.296, z=5.342, rx=175.685, ry=-2.348, rz=115, fatherId=fPrdFrame[0]}
  [587] = {x=-59.909, y=-108.296, z=5.281, rx=175.685, ry=-2.289, rz=115, fatherId=fPrdFrame[0]}
  [588] = {x=-58.425, y=-108.296, z=5.222, rx=175.685, ry=-2.23, rz=115, fatherId=fPrdFrame[0]}
  [589] = {x=-56.942, y=-108.296, z=5.164, rx=175.685, ry=-2.171, rz=115, fatherId=fPrdFrame[0]}
  [590] = {x=-55.459, y=-108.296, z=5.108, rx=175.685, ry=-2.111, rz=115, fatherId=fPrdFrame[0]}
  [591] = {x=-53.975, y=-108.296, z=5.054, rx=175.685, ry=-2.052, rz=115, fatherId=fPrdFrame[0]}
  [592] = {x=-52.492, y=-108.296, z=5.001, rx=175.686, ry=-1.993, rz=115, fatherId=fPrdFrame[0]}
  [593] = {x=-51.008, y=-108.296, z=4.949, rx=175.686, ry=-1.934, rz=115, fatherId=fPrdFrame[0]}
  [594] = {x=-49.525, y=-108.296, z=4.899, rx=175.686, ry=-1.874, rz=115, fatherId=fPrdFrame[0]}
  [595] = {x=-48.041, y=-108.296, z=4.851, rx=175.686, ry=-1.815, rz=115, fatherId=fPrdFrame[0]}
  [596] = {x=-46.558, y=-108.297, z=4.804, rx=175.686, ry=-1.756, rz=115, fatherId=fPrdFrame[0]}
  [597] = {x=-45.074, y=-108.297, z=4.759, rx=175.686, ry=-1.697, rz=115, fatherId=fPrdFrame[0]}
  [598] = {x=-43.591, y=-108.297, z=4.715, rx=175.686, ry=-1.638, rz=115, fatherId=fPrdFrame[0]}
  [599] = {x=-42.107, y=-108.297, z=4.673, rx=175.687, ry=-1.578, rz=115, fatherId=fPrdFrame[0]}
  [600] = {x=-40.624, y=-108.297, z=4.633, rx=175.687, ry=-1.519, rz=115, fatherId=fPrdFrame[0]}
  [601] = {x=-39.14, y=-108.297, z=4.594, rx=175.687, ry=-1.46, rz=115, fatherId=fPrdFrame[0]}
  [602] = {x=-37.657, y=-108.297, z=4.556, rx=175.687, ry=-1.401, rz=115, fatherId=fPrdFrame[0]}
  [603] = {x=-36.173, y=-108.297, z=4.52, rx=175.687, ry=-1.342, rz=115, fatherId=fPrdFrame[0]}
  [604] = {x=-34.69, y=-108.297, z=4.486, rx=175.687, ry=-1.282, rz=115, fatherId=fPrdFrame[0]}
  [605] = {x=-33.206, y=-108.297, z=4.453, rx=175.687, ry=-1.223, rz=115, fatherId=fPrdFrame[0]}
  [606] = {x=-31.723, y=-108.297, z=4.422, rx=175.687, ry=-1.164, rz=115, fatherId=fPrdFrame[0]}
  [607] = {x=-30.239, y=-108.297, z=4.392, rx=175.687, ry=-1.105, rz=115, fatherId=fPrdFrame[0]}
  [608] = {x=-28.756, y=-108.297, z=4.364, rx=175.688, ry=-1.046, rz=115, fatherId=fPrdFrame[0]}
  [609] = {x=-27.273, y=-108.297, z=4.337, rx=175.688, ry=-0.987, rz=115, fatherId=fPrdFrame[0]}
  [610] = {x=-25.789, y=-108.297, z=4.312, rx=175.688, ry=-0.927, rz=115, fatherId=fPrdFrame[0]}
  [611] = {x=-24.306, y=-108.297, z=4.289, rx=175.688, ry=-0.868, rz=115, fatherId=fPrdFrame[0]}
  [612] = {x=-22.822, y=-108.297, z=4.267, rx=175.688, ry=-0.809, rz=115, fatherId=fPrdFrame[0]}
  [613] = {x=-21.339, y=-108.297, z=4.246, rx=175.688, ry=-0.75, rz=115, fatherId=fPrdFrame[0]}
  [614] = {x=-19.855, y=-108.297, z=4.228, rx=175.688, ry=-0.691, rz=115, fatherId=fPrdFrame[0]}
  [615] = {x=-18.372, y=-108.297, z=4.21, rx=175.688, ry=-0.631, rz=115, fatherId=fPrdFrame[0]}
  [616] = {x=-16.888, y=-108.297, z=4.195, rx=175.688, ry=-0.572, rz=115, fatherId=fPrdFrame[0]}
  [617] = {x=-15.405, y=-108.297, z=4.18, rx=175.688, ry=-0.513, rz=115, fatherId=fPrdFrame[0]}
  [618] = {x=-13.921, y=-108.297, z=4.168, rx=175.688, ry=-0.454, rz=115, fatherId=fPrdFrame[0]}
  [619] = {x=-12.438, y=-108.297, z=4.157, rx=175.688, ry=-0.395, rz=115, fatherId=fPrdFrame[0]}
  [620] = {x=-10.954, y=-108.297, z=4.147, rx=175.688, ry=-0.336, rz=115, fatherId=fPrdFrame[0]}
  [621] = {x=-9.471, y=-108.297, z=4.139, rx=175.688, ry=-0.276, rz=115, fatherId=fPrdFrame[0]}
  [622] = {x=-7.987, y=-108.297, z=4.133, rx=175.688, ry=-0.217, rz=115, fatherId=fPrdFrame[0]}
  [623] = {x=-6.504, y=-108.297, z=4.128, rx=175.688, ry=-0.158, rz=115, fatherId=fPrdFrame[0]}
  [624] = {x=-5.02, y=-108.297, z=4.124, rx=175.688, ry=-0.099, rz=115, fatherId=fPrdFrame[0]}
  [625] = {x=-3.537, y=-108.297, z=4.122, rx=175.688, ry=-0.04, rz=115, fatherId=fPrdFrame[0]}
  [626] = {x=-2.053, y=-108.297, z=4.122, rx=175.688, ry=0.02, rz=115, fatherId=fPrdFrame[0]}
  [627] = {x=-0.57, y=-108.297, z=4.123, rx=175.688, ry=0.079, rz=115, fatherId=fPrdFrame[0]}
  [628] = {x=0.913, y=-108.297, z=4.126, rx=175.688, ry=0.138, rz=115, fatherId=fPrdFrame[0]}
  [629] = {x=2.397, y=-108.297, z=4.131, rx=175.688, ry=0.197, rz=115, fatherId=fPrdFrame[0]}
  [630] = {x=3.88, y=-108.297, z=4.137, rx=175.688, ry=0.256, rz=115, fatherId=fPrdFrame[0]}
  [631] = {x=5.364, y=-108.297, z=4.144, rx=175.688, ry=0.315, rz=115, fatherId=fPrdFrame[0]}
  [632] = {x=6.847, y=-108.297, z=4.153, rx=175.688, ry=0.375, rz=115, fatherId=fPrdFrame[0]}
  [633] = {x=8.331, y=-108.297, z=4.164, rx=175.688, ry=0.434, rz=115, fatherId=fPrdFrame[0]}
  [634] = {x=9.814, y=-108.297, z=4.176, rx=175.688, ry=0.493, rz=115, fatherId=fPrdFrame[0]}
  [635] = {x=11.298, y=-108.297, z=4.19, rx=175.688, ry=0.552, rz=115, fatherId=fPrdFrame[0]}
  [636] = {x=12.781, y=-108.297, z=4.205, rx=175.688, ry=0.611, rz=115, fatherId=fPrdFrame[0]}
  [637] = {x=14.265, y=-108.297, z=4.222, rx=175.688, ry=0.67, rz=115, fatherId=fPrdFrame[0]}
  [638] = {x=15.748, y=-108.297, z=4.24, rx=175.688, ry=0.73, rz=115, fatherId=fPrdFrame[0]}
  [639] = {x=17.232, y=-108.297, z=4.26, rx=175.688, ry=0.789, rz=115, fatherId=fPrdFrame[0]}
  [640] = {x=18.715, y=-108.297, z=4.281, rx=175.688, ry=0.848, rz=115, fatherId=fPrdFrame[0]}
  [641] = {x=20.199, y=-108.297, z=4.304, rx=175.688, ry=0.907, rz=115, fatherId=fPrdFrame[0]}
  [642] = {x=21.682, y=-108.297, z=4.329, rx=175.688, ry=0.966, rz=115, fatherId=fPrdFrame[0]}
  [643] = {x=23.166, y=-108.297, z=4.355, rx=175.688, ry=1.026, rz=115, fatherId=fPrdFrame[0]}
  [644] = {x=24.649, y=-108.297, z=4.382, rx=175.687, ry=1.085, rz=115, fatherId=fPrdFrame[0]}
  [645] = {x=26.133, y=-108.297, z=4.412, rx=175.687, ry=1.144, rz=115, fatherId=fPrdFrame[0]}
  [646] = {x=27.616, y=-108.297, z=4.442, rx=175.687, ry=1.203, rz=115, fatherId=fPrdFrame[0]}
  [647] = {x=29.1, y=-108.297, z=4.475, rx=175.687, ry=1.262, rz=115, fatherId=fPrdFrame[0]}
  [648] = {x=30.583, y=-108.297, z=4.508, rx=175.687, ry=1.322, rz=115, fatherId=fPrdFrame[0]}
  [649] = {x=32.066, y=-108.297, z=4.544, rx=175.687, ry=1.381, rz=115, fatherId=fPrdFrame[0]}
  [650] = {x=33.55, y=-108.297, z=4.581, rx=175.687, ry=1.44, rz=115, fatherId=fPrdFrame[0]}
  [651] = {x=35.033, y=-108.297, z=4.619, rx=175.687, ry=1.499, rz=115, fatherId=fPrdFrame[0]}
  [652] = {x=36.517, y=-108.297, z=4.659, rx=175.687, ry=1.558, rz=115, fatherId=fPrdFrame[0]}
  [653] = {x=38, y=-108.297, z=4.701, rx=175.687, ry=1.618, rz=115, fatherId=fPrdFrame[0]}
  [654] = {x=39.484, y=-108.297, z=4.744, rx=175.686, ry=1.677, rz=115, fatherId=fPrdFrame[0]}
  [655] = {x=40.967, y=-108.297, z=4.789, rx=175.686, ry=1.736, rz=115, fatherId=fPrdFrame[0]}
  [656] = {x=42.451, y=-108.296, z=4.835, rx=175.686, ry=1.795, rz=115, fatherId=fPrdFrame[0]}
  [657] = {x=43.934, y=-108.296, z=4.883, rx=175.686, ry=1.854, rz=115, fatherId=fPrdFrame[0]}
  [658] = {x=45.418, y=-108.296, z=4.932, rx=175.686, ry=1.914, rz=115, fatherId=fPrdFrame[0]}
  [659] = {x=46.901, y=-108.296, z=4.983, rx=175.686, ry=1.973, rz=115, fatherId=fPrdFrame[0]}
  [660] = {x=48.385, y=-108.296, z=5.035, rx=175.686, ry=2.032, rz=115, fatherId=fPrdFrame[0]}
  [661] = {x=49.868, y=-108.296, z=5.089, rx=175.685, ry=2.091, rz=115, fatherId=fPrdFrame[0]}
  [662] = {x=51.352, y=-108.296, z=5.145, rx=175.685, ry=2.15, rz=115, fatherId=fPrdFrame[0]}
  [663] = {x=52.835, y=-108.296, z=5.202, rx=175.685, ry=2.21, rz=115, fatherId=fPrdFrame[0]}
  [664] = {x=54.319, y=-108.296, z=5.261, rx=175.685, ry=2.269, rz=115, fatherId=fPrdFrame[0]}
  [665] = {x=55.802, y=-108.296, z=5.321, rx=175.685, ry=2.328, rz=115, fatherId=fPrdFrame[0]}
  [666] = {x=57.286, y=-108.296, z=5.383, rx=175.685, ry=2.387, rz=115, fatherId=fPrdFrame[0]}
  [667] = {x=58.769, y=-108.296, z=5.446, rx=175.684, ry=2.447, rz=115, fatherId=fPrdFrame[0]}
  [668] = {x=60.252, y=-108.296, z=5.511, rx=175.684, ry=2.506, rz=115, fatherId=fPrdFrame[0]}
  [669] = {x=61.736, y=-106.812, z=5.465, rx=175.743, ry=2.565, rz=115, fatherId=fPrdFrame[0]}
  [670] = {x=60.253, y=-106.812, z=5.398, rx=175.743, ry=2.506, rz=115, fatherId=fPrdFrame[0]}
  [671] = {x=58.769, y=-106.812, z=5.333, rx=175.744, ry=2.446, rz=115, fatherId=fPrdFrame[0]}
  [672] = {x=57.286, y=-106.813, z=5.27, rx=175.744, ry=2.387, rz=115, fatherId=fPrdFrame[0]}
  [673] = {x=55.802, y=-106.813, z=5.208, rx=175.744, ry=2.328, rz=115, fatherId=fPrdFrame[0]}
  [674] = {x=54.319, y=-106.813, z=5.148, rx=175.744, ry=2.269, rz=115, fatherId=fPrdFrame[0]}
  [675] = {x=52.835, y=-106.813, z=5.09, rx=175.744, ry=2.209, rz=115, fatherId=fPrdFrame[0]}
  [676] = {x=51.352, y=-106.813, z=5.032, rx=175.744, ry=2.15, rz=115, fatherId=fPrdFrame[0]}
  [677] = {x=49.868, y=-106.813, z=4.977, rx=175.745, ry=2.091, rz=115, fatherId=fPrdFrame[0]}
  [678] = {x=48.385, y=-106.813, z=4.923, rx=175.745, ry=2.032, rz=115, fatherId=fPrdFrame[0]}
  [679] = {x=46.901, y=-106.813, z=4.871, rx=175.745, ry=1.973, rz=115, fatherId=fPrdFrame[0]}
  [680] = {x=45.418, y=-106.813, z=4.82, rx=175.745, ry=1.913, rz=115, fatherId=fPrdFrame[0]}
  [681] = {x=43.934, y=-106.813, z=4.77, rx=175.745, ry=1.854, rz=115, fatherId=fPrdFrame[0]}
  [682] = {x=42.451, y=-106.813, z=4.723, rx=175.745, ry=1.795, rz=115, fatherId=fPrdFrame[0]}
  [683] = {x=40.967, y=-106.813, z=4.676, rx=175.745, ry=1.736, rz=115, fatherId=fPrdFrame[0]}
  [684] = {x=39.484, y=-106.813, z=4.632, rx=175.746, ry=1.677, rz=115, fatherId=fPrdFrame[0]}
  [685] = {x=38, y=-106.813, z=4.588, rx=175.746, ry=1.617, rz=115, fatherId=fPrdFrame[0]}
  [686] = {x=36.517, y=-106.813, z=4.547, rx=175.746, ry=1.558, rz=115, fatherId=fPrdFrame[0]}
  [687] = {x=35.033, y=-106.813, z=4.507, rx=175.746, ry=1.499, rz=115, fatherId=fPrdFrame[0]}
  [688] = {x=33.55, y=-106.813, z=4.468, rx=175.746, ry=1.44, rz=115, fatherId=fPrdFrame[0]}
  [689] = {x=32.066, y=-106.813, z=4.431, rx=175.746, ry=1.381, rz=115, fatherId=fPrdFrame[0]}
  [690] = {x=30.583, y=-106.813, z=4.396, rx=175.746, ry=1.321, rz=115, fatherId=fPrdFrame[0]}
  [691] = {x=29.1, y=-106.813, z=4.362, rx=175.746, ry=1.262, rz=115, fatherId=fPrdFrame[0]}
  [692] = {x=27.616, y=-106.813, z=4.33, rx=175.746, ry=1.203, rz=115, fatherId=fPrdFrame[0]}
  [693] = {x=26.133, y=-106.813, z=4.299, rx=175.747, ry=1.144, rz=115, fatherId=fPrdFrame[0]}
  [694] = {x=24.649, y=-106.813, z=4.27, rx=175.747, ry=1.085, rz=115, fatherId=fPrdFrame[0]}
  [695] = {x=23.166, y=-106.813, z=4.242, rx=175.747, ry=1.026, rz=115, fatherId=fPrdFrame[0]}
  [696] = {x=21.682, y=-106.813, z=4.216, rx=175.747, ry=0.966, rz=115, fatherId=fPrdFrame[0]}
  [697] = {x=20.199, y=-106.813, z=4.192, rx=175.747, ry=0.907, rz=115, fatherId=fPrdFrame[0]}
  [698] = {x=18.715, y=-106.813, z=4.169, rx=175.747, ry=0.848, rz=115, fatherId=fPrdFrame[0]}
  [699] = {x=17.232, y=-106.813, z=4.147, rx=175.747, ry=0.789, rz=115, fatherId=fPrdFrame[0]}
  [700] = {x=15.748, y=-106.813, z=4.128, rx=175.747, ry=0.73, rz=115, fatherId=fPrdFrame[0]}
  [701] = {x=14.265, y=-106.813, z=4.109, rx=175.747, ry=0.67, rz=115, fatherId=fPrdFrame[0]}
  [702] = {x=12.781, y=-106.813, z=4.092, rx=175.747, ry=0.611, rz=115, fatherId=fPrdFrame[0]}
  [703] = {x=11.298, y=-106.813, z=4.077, rx=175.747, ry=0.552, rz=115, fatherId=fPrdFrame[0]}
  [704] = {x=9.814, y=-106.814, z=4.064, rx=175.747, ry=0.493, rz=115, fatherId=fPrdFrame[0]}
  [705] = {x=8.331, y=-106.814, z=4.051, rx=175.747, ry=0.434, rz=115, fatherId=fPrdFrame[0]}
  [706] = {x=6.847, y=-106.814, z=4.041, rx=175.747, ry=0.375, rz=115, fatherId=fPrdFrame[0]}
  [707] = {x=5.364, y=-106.814, z=4.032, rx=175.747, ry=0.315, rz=115, fatherId=fPrdFrame[0]}
  [708] = {x=3.88, y=-106.814, z=4.024, rx=175.747, ry=0.256, rz=115, fatherId=fPrdFrame[0]}
  [709] = {x=2.397, y=-106.814, z=4.018, rx=175.747, ry=0.197, rz=115, fatherId=fPrdFrame[0]}
  [710] = {x=0.913, y=-106.814, z=4.014, rx=175.747, ry=0.138, rz=115, fatherId=fPrdFrame[0]}
  [711] = {x=-0.57, y=-106.814, z=4.011, rx=175.747, ry=0.079, rz=115, fatherId=fPrdFrame[0]}
  [712] = {x=-2.053, y=-106.814, z=4.01, rx=175.747, ry=0.02, rz=115, fatherId=fPrdFrame[0]}
  [713] = {x=-3.537, y=-106.814, z=4.01, rx=175.747, ry=-0.04, rz=115, fatherId=fPrdFrame[0]}
  [714] = {x=-5.02, y=-106.814, z=4.012, rx=175.747, ry=-0.099, rz=115, fatherId=fPrdFrame[0]}
  [715] = {x=-6.504, y=-106.814, z=4.015, rx=175.747, ry=-0.158, rz=115, fatherId=fPrdFrame[0]}
  [716] = {x=-7.987, y=-106.814, z=4.02, rx=175.747, ry=-0.217, rz=115, fatherId=fPrdFrame[0]}
  [717] = {x=-9.471, y=-106.814, z=4.027, rx=175.747, ry=-0.276, rz=115, fatherId=fPrdFrame[0]}
  [718] = {x=-10.954, y=-106.814, z=4.035, rx=175.747, ry=-0.336, rz=115, fatherId=fPrdFrame[0]}
  [719] = {x=-12.438, y=-106.814, z=4.044, rx=175.747, ry=-0.395, rz=115, fatherId=fPrdFrame[0]}
  [720] = {x=-13.921, y=-106.814, z=4.055, rx=175.747, ry=-0.454, rz=115, fatherId=fPrdFrame[0]}
  [721] = {x=-15.405, y=-106.813, z=4.068, rx=175.747, ry=-0.513, rz=115, fatherId=fPrdFrame[0]}
  [722] = {x=-16.888, y=-106.813, z=4.082, rx=175.747, ry=-0.572, rz=115, fatherId=fPrdFrame[0]}
  [723] = {x=-18.372, y=-106.813, z=4.098, rx=175.747, ry=-0.631, rz=115, fatherId=fPrdFrame[0]}
  [724] = {x=-19.855, y=-106.813, z=4.115, rx=175.747, ry=-0.691, rz=115, fatherId=fPrdFrame[0]}
  [725] = {x=-21.339, y=-106.813, z=4.134, rx=175.747, ry=-0.75, rz=115, fatherId=fPrdFrame[0]}
  [726] = {x=-22.822, y=-106.813, z=4.155, rx=175.747, ry=-0.809, rz=115, fatherId=fPrdFrame[0]}
  [727] = {x=-24.306, y=-106.813, z=4.177, rx=175.747, ry=-0.868, rz=115, fatherId=fPrdFrame[0]}
  [728] = {x=-25.789, y=-106.813, z=4.2, rx=175.747, ry=-0.927, rz=115, fatherId=fPrdFrame[0]}
  [729] = {x=-27.273, y=-106.813, z=4.225, rx=175.747, ry=-0.986, rz=115, fatherId=fPrdFrame[0]}
  [730] = {x=-28.756, y=-106.813, z=4.252, rx=175.747, ry=-1.046, rz=115, fatherId=fPrdFrame[0]}
  [731] = {x=-30.239, y=-106.813, z=4.28, rx=175.747, ry=-1.105, rz=115, fatherId=fPrdFrame[0]}
  [732] = {x=-31.723, y=-106.813, z=4.31, rx=175.747, ry=-1.164, rz=115, fatherId=fPrdFrame[0]}
  [733] = {x=-33.206, y=-106.813, z=4.341, rx=175.746, ry=-1.223, rz=115, fatherId=fPrdFrame[0]}
  [734] = {x=-34.69, y=-106.813, z=4.374, rx=175.746, ry=-1.282, rz=115, fatherId=fPrdFrame[0]}
  [735] = {x=-36.173, y=-106.813, z=4.408, rx=175.746, ry=-1.342, rz=115, fatherId=fPrdFrame[0]}
  [736] = {x=-37.657, y=-106.813, z=4.444, rx=175.746, ry=-1.401, rz=115, fatherId=fPrdFrame[0]}
  [737] = {x=-39.14, y=-106.813, z=4.481, rx=175.746, ry=-1.46, rz=115, fatherId=fPrdFrame[0]}
  [738] = {x=-40.624, y=-106.813, z=4.52, rx=175.746, ry=-1.519, rz=115, fatherId=fPrdFrame[0]}
  [739] = {x=-42.107, y=-106.813, z=4.561, rx=175.746, ry=-1.578, rz=115, fatherId=fPrdFrame[0]}
  [740] = {x=-43.591, y=-106.813, z=4.603, rx=175.746, ry=-1.638, rz=115, fatherId=fPrdFrame[0]}
  [741] = {x=-45.074, y=-106.813, z=4.647, rx=175.746, ry=-1.697, rz=115, fatherId=fPrdFrame[0]}
  [742] = {x=-46.558, y=-106.813, z=4.692, rx=175.745, ry=-1.756, rz=115, fatherId=fPrdFrame[0]}
  [743] = {x=-48.041, y=-106.813, z=4.739, rx=175.745, ry=-1.815, rz=115, fatherId=fPrdFrame[0]}
  [744] = {x=-49.525, y=-106.813, z=4.787, rx=175.745, ry=-1.874, rz=115, fatherId=fPrdFrame[0]}
  [745] = {x=-51.008, y=-106.813, z=4.837, rx=175.745, ry=-1.934, rz=115, fatherId=fPrdFrame[0]}
  [746] = {x=-52.492, y=-106.813, z=4.888, rx=175.745, ry=-1.993, rz=115, fatherId=fPrdFrame[0]}
  [747] = {x=-53.975, y=-106.813, z=4.941, rx=175.745, ry=-2.052, rz=115, fatherId=fPrdFrame[0]}
  [748] = {x=-55.459, y=-106.813, z=4.996, rx=175.745, ry=-2.111, rz=115, fatherId=fPrdFrame[0]}
  [749] = {x=-56.942, y=-106.813, z=5.052, rx=175.744, ry=-2.17, rz=115, fatherId=fPrdFrame[0]}
  [750] = {x=-58.426, y=-106.813, z=5.109, rx=175.744, ry=-2.23, rz=115, fatherId=fPrdFrame[0]}
  [751] = {x=-59.909, y=-106.813, z=5.169, rx=175.744, ry=-2.289, rz=115, fatherId=fPrdFrame[0]}
  [752] = {x=-61.392, y=-106.813, z=5.229, rx=175.744, ry=-2.348, rz=115, fatherId=fPrdFrame[0]}
  [753] = {x=-62.876, y=-106.813, z=5.292, rx=175.744, ry=-2.407, rz=115, fatherId=fPrdFrame[0]}
  [754] = {x=-64.359, y=-106.812, z=5.355, rx=175.743, ry=-2.466, rz=115, fatherId=fPrdFrame[0]}
  [755] = {x=-65.843, y=-106.812, z=5.421, rx=175.743, ry=-2.526, rz=115, fatherId=fPrdFrame[0]}
  [756] = {x=-67.326, y=-106.812, z=5.488, rx=175.743, ry=-2.585, rz=115, fatherId=fPrdFrame[0]}
  [757] = {x=-70.293, y=-105.329, z=5.515, rx=175.802, ry=-2.703, rz=115, fatherId=fPrdFrame[0]}
  [758] = {x=-68.81, y=-105.329, z=5.445, rx=175.802, ry=-2.644, rz=115, fatherId=fPrdFrame[0]}
  [759] = {x=-67.326, y=-105.329, z=5.377, rx=175.802, ry=-2.585, rz=115, fatherId=fPrdFrame[0]}
  [760] = {x=-65.843, y=-105.329, z=5.31, rx=175.803, ry=-2.526, rz=115, fatherId=fPrdFrame[0]}
  [761] = {x=-64.359, y=-105.329, z=5.245, rx=175.803, ry=-2.466, rz=115, fatherId=fPrdFrame[0]}
  [762] = {x=-62.876, y=-105.329, z=5.181, rx=175.803, ry=-2.407, rz=115, fatherId=fPrdFrame[0]}
  [763] = {x=-61.393, y=-105.329, z=5.118, rx=175.803, ry=-2.348, rz=115, fatherId=fPrdFrame[0]}
  [764] = {x=-59.909, y=-105.329, z=5.058, rx=175.803, ry=-2.289, rz=115, fatherId=fPrdFrame[0]}
  [765] = {x=-58.426, y=-105.329, z=4.999, rx=175.803, ry=-2.229, rz=115, fatherId=fPrdFrame[0]}
  [766] = {x=-56.942, y=-105.329, z=4.941, rx=175.804, ry=-2.17, rz=115, fatherId=fPrdFrame[0]}
  [767] = {x=-55.459, y=-105.329, z=4.885, rx=175.804, ry=-2.111, rz=115, fatherId=fPrdFrame[0]}
  [768] = {x=-53.975, y=-105.329, z=4.83, rx=175.804, ry=-2.052, rz=115, fatherId=fPrdFrame[0]}
  [769] = {x=-52.492, y=-105.329, z=4.777, rx=175.804, ry=-1.993, rz=115, fatherId=fPrdFrame[0]}
  [770] = {x=-51.008, y=-105.329, z=4.726, rx=175.804, ry=-1.933, rz=115, fatherId=fPrdFrame[0]}
  [771] = {x=-49.525, y=-105.329, z=4.676, rx=175.804, ry=-1.874, rz=115, fatherId=fPrdFrame[0]}
  [772] = {x=-48.041, y=-105.329, z=4.628, rx=175.804, ry=-1.815, rz=115, fatherId=fPrdFrame[0]}
  [773] = {x=-46.558, y=-105.329, z=4.581, rx=175.805, ry=-1.756, rz=115, fatherId=fPrdFrame[0]}
  [774] = {x=-45.074, y=-105.33, z=4.536, rx=175.805, ry=-1.697, rz=115, fatherId=fPrdFrame[0]}
  [775] = {x=-43.591, y=-105.33, z=4.492, rx=175.805, ry=-1.637, rz=115, fatherId=fPrdFrame[0]}
  [776] = {x=-42.107, y=-105.33, z=4.45, rx=175.805, ry=-1.578, rz=115, fatherId=fPrdFrame[0]}
  [777] = {x=-40.624, y=-105.33, z=4.409, rx=175.805, ry=-1.519, rz=115, fatherId=fPrdFrame[0]}
  [778] = {x=-39.14, y=-105.33, z=4.37, rx=175.805, ry=-1.46, rz=115, fatherId=fPrdFrame[0]}
  [779] = {x=-37.657, y=-105.33, z=4.333, rx=175.805, ry=-1.401, rz=115, fatherId=fPrdFrame[0]}
  [780] = {x=-36.173, y=-105.33, z=4.297, rx=175.805, ry=-1.341, rz=115, fatherId=fPrdFrame[0]}
  [781] = {x=-34.69, y=-105.33, z=4.263, rx=175.806, ry=-1.282, rz=115, fatherId=fPrdFrame[0]}
  [782] = {x=-33.206, y=-105.33, z=4.23, rx=175.806, ry=-1.223, rz=115, fatherId=fPrdFrame[0]}
  [783] = {x=-31.723, y=-105.33, z=4.199, rx=175.806, ry=-1.164, rz=115, fatherId=fPrdFrame[0]}
  [784] = {x=-30.24, y=-105.33, z=4.169, rx=175.806, ry=-1.105, rz=115, fatherId=fPrdFrame[0]}
  [785] = {x=-28.756, y=-105.33, z=4.141, rx=175.806, ry=-1.046, rz=115, fatherId=fPrdFrame[0]}
  [786] = {x=-27.273, y=-105.33, z=4.114, rx=175.806, ry=-0.986, rz=115, fatherId=fPrdFrame[0]}
  [787] = {x=-25.789, y=-105.33, z=4.089, rx=175.806, ry=-0.927, rz=115, fatherId=fPrdFrame[0]}
  [788] = {x=-24.306, y=-105.33, z=4.066, rx=175.806, ry=-0.868, rz=115, fatherId=fPrdFrame[0]}
  [789] = {x=-22.822, y=-105.33, z=4.044, rx=175.806, ry=-0.809, rz=115, fatherId=fPrdFrame[0]}
  [790] = {x=-21.339, y=-105.33, z=4.023, rx=175.806, ry=-0.75, rz=115, fatherId=fPrdFrame[0]}
  [791] = {x=-19.855, y=-105.33, z=4.005, rx=175.806, ry=-0.691, rz=115, fatherId=fPrdFrame[0]}
  [792] = {x=-18.372, y=-105.33, z=3.987, rx=175.806, ry=-0.631, rz=115, fatherId=fPrdFrame[0]}
  [793] = {x=-16.888, y=-105.33, z=3.971, rx=175.806, ry=-0.572, rz=115, fatherId=fPrdFrame[0]}
  [794] = {x=-15.405, y=-105.33, z=3.957, rx=175.806, ry=-0.513, rz=115, fatherId=fPrdFrame[0]}
  [795] = {x=-13.921, y=-105.33, z=3.945, rx=175.806, ry=-0.454, rz=115, fatherId=fPrdFrame[0]}
  [796] = {x=-12.438, y=-105.33, z=3.934, rx=175.806, ry=-0.395, rz=115, fatherId=fPrdFrame[0]}
  [797] = {x=-10.954, y=-105.33, z=3.924, rx=175.807, ry=-0.335, rz=115, fatherId=fPrdFrame[0]}
  [798] = {x=-9.471, y=-105.33, z=3.916, rx=175.807, ry=-0.276, rz=115, fatherId=fPrdFrame[0]}
  [799] = {x=-7.987, y=-105.33, z=3.909, rx=175.807, ry=-0.217, rz=115, fatherId=fPrdFrame[0]}
  [800] = {x=-6.504, y=-105.33, z=3.905, rx=175.807, ry=-0.158, rz=115, fatherId=fPrdFrame[0]}
  [801] = {x=-5.02, y=-105.33, z=3.901, rx=175.807, ry=-0.099, rz=115, fatherId=fPrdFrame[0]}
  [802] = {x=-3.537, y=-105.33, z=3.899, rx=175.807, ry=-0.04, rz=115, fatherId=fPrdFrame[0]}
  [803] = {x=-2.053, y=-105.33, z=3.899, rx=175.807, ry=0.02, rz=115, fatherId=fPrdFrame[0]}
  [804] = {x=-0.57, y=-105.33, z=3.9, rx=175.807, ry=0.079, rz=115, fatherId=fPrdFrame[0]}
  [805] = {x=0.914, y=-105.33, z=3.903, rx=175.807, ry=0.138, rz=115, fatherId=fPrdFrame[0]}
  [806] = {x=2.397, y=-105.33, z=3.908, rx=175.807, ry=0.197, rz=115, fatherId=fPrdFrame[0]}
  [807] = {x=3.88, y=-105.33, z=3.914, rx=175.807, ry=0.256, rz=115, fatherId=fPrdFrame[0]}
  [808] = {x=5.364, y=-105.33, z=3.921, rx=175.807, ry=0.315, rz=115, fatherId=fPrdFrame[0]}
  [809] = {x=6.847, y=-105.33, z=3.93, rx=175.806, ry=0.375, rz=115, fatherId=fPrdFrame[0]}
  [810] = {x=8.331, y=-105.33, z=3.941, rx=175.806, ry=0.434, rz=115, fatherId=fPrdFrame[0]}
  [811] = {x=9.814, y=-105.33, z=3.953, rx=175.806, ry=0.493, rz=115, fatherId=fPrdFrame[0]}
  [812] = {x=11.298, y=-105.33, z=3.966, rx=175.806, ry=0.552, rz=115, fatherId=fPrdFrame[0]}
  [813] = {x=12.781, y=-105.33, z=3.982, rx=175.806, ry=0.611, rz=115, fatherId=fPrdFrame[0]}
  [814] = {x=14.265, y=-105.33, z=3.998, rx=175.806, ry=0.67, rz=115, fatherId=fPrdFrame[0]}
  [815] = {x=15.748, y=-105.33, z=4.017, rx=175.806, ry=0.73, rz=115, fatherId=fPrdFrame[0]}
  [816] = {x=17.232, y=-105.33, z=4.037, rx=175.806, ry=0.789, rz=115, fatherId=fPrdFrame[0]}
  [817] = {x=18.715, y=-105.33, z=4.058, rx=175.806, ry=0.848, rz=115, fatherId=fPrdFrame[0]}
  [818] = {x=20.199, y=-105.33, z=4.081, rx=175.806, ry=0.907, rz=115, fatherId=fPrdFrame[0]}
  [819] = {x=21.682, y=-105.33, z=4.106, rx=175.806, ry=0.966, rz=115, fatherId=fPrdFrame[0]}
  [820] = {x=23.166, y=-105.33, z=4.132, rx=175.806, ry=1.025, rz=115, fatherId=fPrdFrame[0]}
  [821] = {x=24.649, y=-105.33, z=4.159, rx=175.806, ry=1.085, rz=115, fatherId=fPrdFrame[0]}
  [822] = {x=26.133, y=-105.33, z=4.188, rx=175.806, ry=1.144, rz=115, fatherId=fPrdFrame[0]}
  [823] = {x=27.616, y=-105.33, z=4.219, rx=175.806, ry=1.203, rz=115, fatherId=fPrdFrame[0]}
  [824] = {x=29.1, y=-105.33, z=4.251, rx=175.806, ry=1.262, rz=115, fatherId=fPrdFrame[0]}
  [825] = {x=30.583, y=-105.33, z=4.285, rx=175.805, ry=1.321, rz=115, fatherId=fPrdFrame[0]}
  [826] = {x=32.067, y=-105.33, z=4.321, rx=175.805, ry=1.381, rz=115, fatherId=fPrdFrame[0]}
  [827] = {x=33.55, y=-105.33, z=4.358, rx=175.805, ry=1.44, rz=115, fatherId=fPrdFrame[0]}
  [828] = {x=35.033, y=-105.33, z=4.396, rx=175.805, ry=1.499, rz=115, fatherId=fPrdFrame[0]}
  [829] = {x=36.517, y=-105.33, z=4.436, rx=175.805, ry=1.558, rz=115, fatherId=fPrdFrame[0]}
  [830] = {x=38, y=-105.33, z=4.478, rx=175.805, ry=1.617, rz=115, fatherId=fPrdFrame[0]}
  [831] = {x=39.484, y=-105.33, z=4.521, rx=175.805, ry=1.676, rz=115, fatherId=fPrdFrame[0]}
  [832] = {x=40.967, y=-105.329, z=4.565, rx=175.805, ry=1.736, rz=115, fatherId=fPrdFrame[0]}
  [833] = {x=42.451, y=-105.329, z=4.612, rx=175.805, ry=1.795, rz=115, fatherId=fPrdFrame[0]}
  [834] = {x=43.934, y=-105.329, z=4.659, rx=175.804, ry=1.854, rz=115, fatherId=fPrdFrame[0]}
  [835] = {x=45.418, y=-105.329, z=4.709, rx=175.804, ry=1.913, rz=115, fatherId=fPrdFrame[0]}
  [836] = {x=46.901, y=-105.329, z=4.76, rx=175.804, ry=1.972, rz=115, fatherId=fPrdFrame[0]}
  [837] = {x=48.385, y=-105.329, z=4.812, rx=175.804, ry=2.032, rz=115, fatherId=fPrdFrame[0]}
  [838] = {x=49.868, y=-105.329, z=4.866, rx=175.804, ry=2.091, rz=115, fatherId=fPrdFrame[0]}
  [839] = {x=51.352, y=-105.329, z=4.922, rx=175.804, ry=2.15, rz=115, fatherId=fPrdFrame[0]}
  [840] = {x=52.835, y=-105.329, z=4.979, rx=175.803, ry=2.209, rz=115, fatherId=fPrdFrame[0]}
  [841] = {x=54.319, y=-105.329, z=5.037, rx=175.803, ry=2.268, rz=115, fatherId=fPrdFrame[0]}
  [842] = {x=55.802, y=-105.329, z=5.098, rx=175.803, ry=2.328, rz=115, fatherId=fPrdFrame[0]}
  [843] = {x=57.286, y=-105.329, z=5.159, rx=175.803, ry=2.387, rz=115, fatherId=fPrdFrame[0]}
  [844] = {x=58.769, y=-105.329, z=5.223, rx=175.803, ry=2.446, rz=115, fatherId=fPrdFrame[0]}
  [845] = {x=60.253, y=-105.329, z=5.287, rx=175.803, ry=2.505, rz=115, fatherId=fPrdFrame[0]}
  [846] = {x=61.736, y=-105.329, z=5.354, rx=175.802, ry=2.565, rz=115, fatherId=fPrdFrame[0]}
  [847] = {x=63.22, y=-105.329, z=5.422, rx=175.802, ry=2.624, rz=115, fatherId=fPrdFrame[0]}
  [848] = {x=64.703, y=-105.329, z=5.491, rx=175.802, ry=2.683, rz=115, fatherId=fPrdFrame[0]}
  [849] = {x=67.67, y=-103.845, z=5.526, rx=175.861, ry=2.801, rz=115, fatherId=fPrdFrame[0]}
  [850] = {x=66.187, y=-103.845, z=5.453, rx=175.861, ry=2.742, rz=115, fatherId=fPrdFrame[0]}
  [851] = {x=64.703, y=-103.845, z=5.382, rx=175.861, ry=2.683, rz=115, fatherId=fPrdFrame[0]}
  [852] = {x=63.22, y=-103.845, z=5.313, rx=175.861, ry=2.624, rz=115, fatherId=fPrdFrame[0]}
  [853] = {x=61.736, y=-103.845, z=5.245, rx=175.862, ry=2.564, rz=115, fatherId=fPrdFrame[0]}
  [854] = {x=60.253, y=-103.845, z=5.178, rx=175.862, ry=2.505, rz=115, fatherId=fPrdFrame[0]}
  [855] = {x=58.769, y=-103.845, z=5.113, rx=175.862, ry=2.446, rz=115, fatherId=fPrdFrame[0]}
  [856] = {x=57.286, y=-103.846, z=5.05, rx=175.862, ry=2.387, rz=115, fatherId=fPrdFrame[0]}
  [857] = {x=55.802, y=-103.846, z=4.988, rx=175.862, ry=2.328, rz=115, fatherId=fPrdFrame[0]}
  [858] = {x=54.319, y=-103.846, z=4.928, rx=175.863, ry=2.268, rz=115, fatherId=fPrdFrame[0]}
  [859] = {x=52.835, y=-103.846, z=4.869, rx=175.863, ry=2.209, rz=115, fatherId=fPrdFrame[0]}
  [860] = {x=51.352, y=-103.846, z=4.812, rx=175.863, ry=2.15, rz=115, fatherId=fPrdFrame[0]}
  [861] = {x=49.868, y=-103.846, z=4.757, rx=175.863, ry=2.091, rz=115, fatherId=fPrdFrame[0]}
  [862] = {x=48.385, y=-103.846, z=4.703, rx=175.863, ry=2.032, rz=115, fatherId=fPrdFrame[0]}
  [863] = {x=46.901, y=-103.846, z=4.65, rx=175.863, ry=1.972, rz=115, fatherId=fPrdFrame[0]}
  [864] = {x=45.418, y=-103.846, z=4.6, rx=175.863, ry=1.913, rz=115, fatherId=fPrdFrame[0]}
  [865] = {x=43.934, y=-103.846, z=4.55, rx=175.864, ry=1.854, rz=115, fatherId=fPrdFrame[0]}
  [866] = {x=42.451, y=-103.846, z=4.502, rx=175.864, ry=1.795, rz=115, fatherId=fPrdFrame[0]}
  [867] = {x=40.967, y=-103.846, z=4.456, rx=175.864, ry=1.736, rz=115, fatherId=fPrdFrame[0]}
  [868] = {x=39.484, y=-103.846, z=4.412, rx=175.864, ry=1.676, rz=115, fatherId=fPrdFrame[0]}
  [869] = {x=38, y=-103.846, z=4.368, rx=175.864, ry=1.617, rz=115, fatherId=fPrdFrame[0]}
  [870] = {x=36.517, y=-103.846, z=4.327, rx=175.864, ry=1.558, rz=115, fatherId=fPrdFrame[0]}
  [871] = {x=35.034, y=-103.846, z=4.287, rx=175.864, ry=1.499, rz=115, fatherId=fPrdFrame[0]}
  [872] = {x=33.55, y=-103.846, z=4.248, rx=175.864, ry=1.44, rz=115, fatherId=fPrdFrame[0]}
  [873] = {x=32.067, y=-103.846, z=4.211, rx=175.865, ry=1.38, rz=115, fatherId=fPrdFrame[0]}
  [874] = {x=30.583, y=-103.846, z=4.176, rx=175.865, ry=1.321, rz=115, fatherId=fPrdFrame[0]}
  [875] = {x=29.1, y=-103.846, z=4.142, rx=175.865, ry=1.262, rz=115, fatherId=fPrdFrame[0]}
  [876] = {x=27.616, y=-103.846, z=4.11, rx=175.865, ry=1.203, rz=115, fatherId=fPrdFrame[0]}
  [877] = {x=26.133, y=-103.846, z=4.079, rx=175.865, ry=1.144, rz=115, fatherId=fPrdFrame[0]}
  [878] = {x=24.649, y=-103.846, z=4.05, rx=175.865, ry=1.085, rz=115, fatherId=fPrdFrame[0]}
  [879] = {x=23.166, y=-103.846, z=4.022, rx=175.865, ry=1.025, rz=115, fatherId=fPrdFrame[0]}
  [880] = {x=21.682, y=-103.846, z=3.996, rx=175.865, ry=0.966, rz=115, fatherId=fPrdFrame[0]}
  [881] = {x=20.199, y=-103.846, z=3.972, rx=175.865, ry=0.907, rz=115, fatherId=fPrdFrame[0]}
  [882] = {x=18.715, y=-103.846, z=3.949, rx=175.865, ry=0.848, rz=115, fatherId=fPrdFrame[0]}
  [883] = {x=17.232, y=-103.846, z=3.927, rx=175.865, ry=0.789, rz=115, fatherId=fPrdFrame[0]}
  [884] = {x=15.748, y=-103.846, z=3.908, rx=175.865, ry=0.73, rz=115, fatherId=fPrdFrame[0]}
  [885] = {x=14.265, y=-103.846, z=3.889, rx=175.865, ry=0.67, rz=115, fatherId=fPrdFrame[0]}
  [886] = {x=12.781, y=-103.846, z=3.872, rx=175.866, ry=0.611, rz=115, fatherId=fPrdFrame[0]}
  [887] = {x=11.298, y=-103.846, z=3.857, rx=175.866, ry=0.552, rz=115, fatherId=fPrdFrame[0]}
  [888] = {x=9.814, y=-103.846, z=3.844, rx=175.866, ry=0.493, rz=115, fatherId=fPrdFrame[0]}
  [889] = {x=8.331, y=-103.846, z=3.831, rx=175.866, ry=0.434, rz=115, fatherId=fPrdFrame[0]}
  [890] = {x=6.847, y=-103.846, z=3.821, rx=175.866, ry=0.375, rz=115, fatherId=fPrdFrame[0]}
  [891] = {x=5.364, y=-103.846, z=3.812, rx=175.866, ry=0.315, rz=115, fatherId=fPrdFrame[0]}
  [892] = {x=3.88, y=-103.846, z=3.804, rx=175.866, ry=0.256, rz=115, fatherId=fPrdFrame[0]}
  [893] = {x=2.397, y=-103.846, z=3.798, rx=175.866, ry=0.197, rz=115, fatherId=fPrdFrame[0]}
  [894] = {x=0.914, y=-103.846, z=3.794, rx=175.866, ry=0.138, rz=115, fatherId=fPrdFrame[0]}
  [895] = {x=-0.57, y=-103.847, z=3.791, rx=175.866, ry=0.079, rz=115, fatherId=fPrdFrame[0]}
  [896] = {x=-2.053, y=-103.847, z=3.79, rx=175.866, ry=0.02, rz=115, fatherId=fPrdFrame[0]}
  [897] = {x=-3.537, y=-103.847, z=3.79, rx=175.866, ry=-0.04, rz=115, fatherId=fPrdFrame[0]}
  [898] = {x=-5.02, y=-103.847, z=3.792, rx=175.866, ry=-0.099, rz=115, fatherId=fPrdFrame[0]}
  [899] = {x=-6.504, y=-103.846, z=3.795, rx=175.866, ry=-0.158, rz=115, fatherId=fPrdFrame[0]}
  [900] = {x=-7.987, y=-103.846, z=3.8, rx=175.866, ry=-0.217, rz=115, fatherId=fPrdFrame[0]}
  [901] = {x=-9.471, y=-103.846, z=3.807, rx=175.866, ry=-0.276, rz=115, fatherId=fPrdFrame[0]}
  [902] = {x=8.415, y=-28.247, z=13.928, rx=178.358, ry=0.489, rz=135.188, fatherId=fPrdFrame[0]}
  [903] = {x=10.248, y=-27.664, z=13.929, rx=178.392, ry=0.595, rz=135.189, fatherId=fPrdFrame[0]}
  [904] = {x=12.039, y=-26.966, z=13.93, rx=178.433, ry=0.7, rz=135.19, fatherId=fPrdFrame[0]}
  [905] = {x=13.569, y=-26.259, z=13.931, rx=178.475, ry=0.791, rz=135.191, fatherId=fPrdFrame[0]}
  [906] = {x=15.262, y=-25.345, z=13.932, rx=178.527, ry=0.887, rz=135.192, fatherId=fPrdFrame[0]}
  [907] = {x=16.891, y=-24.323, z=13.933, rx=178.586, ry=0.981, rz=135.193, fatherId=fPrdFrame[0]}
  [908] = {x=18.449, y=-23.197, z=13.933, rx=178.652, ry=1.072, rz=135.193, fatherId=fPrdFrame[0]}
  [909] = {x=19.411, y=-22.42, z=13.934, rx=178.697, ry=1.128, rz=135.194, fatherId=fPrdFrame[0]}
  [910] = {x=20.839, y=-21.132, z=13.935, rx=178.772, ry=1.211, rz=135.194, fatherId=fPrdFrame[0]}
  [911] = {x=22.179, y=-19.753, z=13.935, rx=178.852, ry=1.289, rz=135.194, fatherId=fPrdFrame[0]}
  [912] = {x=23.426, y=-18.29, z=13.936, rx=178.937, ry=1.361, rz=135.193, fatherId=fPrdFrame[0]}
  [913] = {x=24.117, y=-17.389, z=13.936, rx=178.99, ry=1.402, rz=135.193, fatherId=fPrdFrame[0]}
  [914] = {x=25.205, y=-15.803, z=13.937, rx=179.081, ry=1.465, rz=135.192, fatherId=fPrdFrame[0]}
  [915] = {x=25.801, y=-14.829, z=13.937, rx=179.138, ry=1.5, rz=135.192, fatherId=fPrdFrame[0]}
  [916] = {x=26.718, y=-13.139, z=13.938, rx=179.236, ry=1.553, rz=135.191, fatherId=fPrdFrame[0]}
  [917] = {x=27.214, y=-12.1, z=13.938, rx=179.297, ry=1.582, rz=135.19, fatherId=fPrdFrame[0]}
  [918] = {x=27.95, y=-10.324, z=13.938, rx=179.4, ry=1.624, rz=135.189, fatherId=fPrdFrame[0]}
  [919] = {x=28.333, y=-9.246, z=13.938, rx=179.457, ry=1.645, rz=135.189, fatherId=fPrdFrame[0]}
  [920] = {x=28.783, y=-7.761, z=13.939, rx=179.549, ry=1.673, rz=135.187, fatherId=fPrdFrame[0]}
  [921] = {x=29.154, y=-6.252, z=13.939, rx=179.637, ry=1.694, rz=135.186, fatherId=fPrdFrame[0]}
  [922] = {x=29.445, y=-4.726, z=13.939, rx=179.725, ry=1.711, rz=135.185, fatherId=fPrdFrame[0]}
  [923] = {x=29.657, y=-3.159, z=13.939, rx=179.816, ry=1.723, rz=135.183, fatherId=fPrdFrame[0]}
  [924] = {x=29.784, y=-1.581, z=13.939, rx=179.908, ry=1.731, rz=135.182, fatherId=fPrdFrame[0]}
  [925] = {x=29.826, z=13.939, rx=180, ry=1.734, rz=135.181, fatherId=fPrdFrame[0]}
  [926] = {x=29.765, y=1.922, z=13.939, rx=-179.888, ry=1.73, rz=135.179, fatherId=fPrdFrame[0]}
  [927] = {x=29.581, y=3.836, z=13.939, rx=-179.777, ry=1.719, rz=135.177, fatherId=fPrdFrame[0]}
  [928] = {x=29.306, y=5.586, z=13.939, rx=-179.675, ry=1.703, rz=135.176, fatherId=fPrdFrame[0]}
  [929] = {x=28.893, y=7.464, z=13.94, rx=-179.566, ry=1.679, rz=135.174, fatherId=fPrdFrame[0]}
  [930] = {x=28.361, y=9.311, z=13.94, rx=-179.459, ry=1.648, rz=135.173, fatherId=fPrdFrame[0]}
  [931] = {x=27.769, y=10.975, z=13.94, rx=-179.362, ry=1.614, rz=135.172, fatherId=fPrdFrame[0]}
  [932] = {x=27.016, y=12.745, z=13.941, rx=-179.259, ry=1.57, rz=135.171, fatherId=fPrdFrame[0]}
  [933] = {x=26.153, y=14.463, z=13.941, rx=-179.159, ry=1.52, rz=135.17, fatherId=fPrdFrame[0]}
  [934] = {x=25.263, y=15.998, z=13.941, rx=-179.072, ry=1.47, rz=135.169, fatherId=fPrdFrame[0]}
  [935] = {x=24.509, y=17.155, z=13.942, rx=-179.003, ry=1.424, rz=135.168, fatherId=fPrdFrame[0]}
  [936] = {x=23.704, y=18.278, z=13.942, rx=-178.938, ry=1.377, rz=135.168, fatherId=fPrdFrame[0]}
  [937] = {x=22.85, y=19.362, z=13.943, rx=-178.871, ry=1.324, rz=135.168, fatherId=fPrdFrame[0]}
  [938] = {x=21.579, y=20.806, z=13.943, rx=-178.791, ry=1.253, rz=135.167, fatherId=fPrdFrame[0]}
  [939] = {x=20.219, y=22.165, z=13.944, rx=-178.712, ry=1.174, rz=135.168, fatherId=fPrdFrame[0]}
  [940] = {x=18.775, y=23.434, z=13.945, rx=-178.639, ry=1.09, rz=135.168, fatherId=fPrdFrame[0]}
  [941] = {x=17.252, y=24.608, z=13.945, rx=-178.571, ry=1.002, rz=135.168, fatherId=fPrdFrame[0]}
  [942] = {x=15.656, y=25.681, z=13.946, rx=-178.508, ry=0.909, rz=135.169, fatherId=fPrdFrame[0]}
  [943] = {x=13.996, y=26.651, z=13.947, rx=-178.452, ry=0.813, rz=135.17, fatherId=fPrdFrame[0]}
  [944] = {x=12.277, y=27.512, z=13.948, rx=-178.402, ry=0.713, rz=135.171, fatherId=fPrdFrame[0]}
  [945] = {x=10.506, y=28.262, z=13.949, rx=-178.358, ry=0.61, rz=135.172, fatherId=fPrdFrame[0]}
  [946] = {x=8.967, y=28.811, z=13.95, rx=-178.326, ry=0.521, rz=135.173, fatherId=fPrdFrame[0]}
  [947] = {x=7.121, y=29.35, z=13.95, rx=-178.294, ry=0.414, rz=135.175, fatherId=fPrdFrame[0]}
  [948] = {x=5.245, y=29.772, z=13.951, rx=-178.27, ry=0.305, rz=135.176, fatherId=fPrdFrame[0]}
  [949] = {x=3.985, y=29.986, z=13.952, rx=-178.257, ry=0.232, rz=135.177, fatherId=fPrdFrame[0]}
  [950] = {x=2.076, y=30.21, z=13.953, rx=-178.244, ry=0.121, rz=135.179, fatherId=fPrdFrame[0]}
  [951] = {x=0.156, y=30.314, z=13.954, rx=-178.238, ry=0.009, rz=135.181, fatherId=fPrdFrame[0]}
  [952] = {x=-1.116, y=30.317, z=13.955, rx=-178.238, ry=-0.065, rz=135.182, fatherId=fPrdFrame[0]}
  [953] = {x=-3.036, y=30.219, z=13.956, rx=-178.244, ry=-0.176, rz=135.183, fatherId=fPrdFrame[0]}
  [954] = {x=-4.946, y=30.001, z=13.956, rx=-178.257, ry=-0.287, rz=135.185, fatherId=fPrdFrame[0]}
  [955] = {x=-6.235, y=29.783, z=13.957, rx=-178.27, ry=-0.362, rz=135.186, fatherId=fPrdFrame[0]}
  [956] = {x=-8.112, y=29.364, z=13.958, rx=-178.294, ry=-0.47, rz=135.188, fatherId=fPrdFrame[0]}
  [957] = {x=-9.957, y=28.824, z=13.959, rx=-178.326, ry=-0.578, rz=135.189, fatherId=fPrdFrame[0]}
  [958] = {x=-11.221, y=28.379, z=13.96, rx=-178.352, ry=-0.652, rz=135.19, fatherId=fPrdFrame[0]}
  [959] = {x=-12.432, y=27.891, z=13.96, rx=-178.38, ry=-0.722, rz=135.191, fatherId=fPrdFrame[0]}
  [960] = {x=-13.641, y=27.341, z=13.961, rx=-178.412, ry=-0.792, rz=135.192, fatherId=fPrdFrame[0]}
  [961] = {x=-14.824, y=26.737, z=13.961, rx=-178.447, ry=-0.861, rz=135.192, fatherId=fPrdFrame[0]}
  [962] = {x=-15.977, y=26.083, z=13.962, rx=-178.488, ry=-0.933, rz=135.193, fatherId=fPrdFrame[0]}
  [963] = {x=-17.597, y=25.045, z=13.963, rx=-178.545, ry=-1.022, rz=135.194, fatherId=fPrdFrame[0]}
  [964] = {x=-19.147, y=23.907, z=13.964, rx=-178.611, ry=-1.112, rz=135.194, fatherId=fPrdFrame[0]}
  [965] = {x=-20.434, y=22.841, z=13.964, rx=-178.673, ry=-1.187, rz=135.194, fatherId=fPrdFrame[0]}
  [966] = {x=-21.841, y=21.53, z=13.965, rx=-178.749, ry=-1.269, rz=135.195, fatherId=fPrdFrame[0]}
  [967] = {x=-23.162, y=20.134, z=13.966, rx=-178.83, ry=-1.346, rz=135.194, fatherId=fPrdFrame[0]}
  [968] = {x=-24.251, y=18.835, z=13.966, rx=-178.905, ry=-1.409, rz=135.194, fatherId=fPrdFrame[0]}
  [969] = {x=-25.089, y=17.724, z=13.966, rx=-178.97, ry=-1.458, rz=135.194, fatherId=fPrdFrame[0]}
  [970] = {x=-25.866, y=16.591, z=13.967, rx=-179.035, ry=-1.503, rz=135.193, fatherId=fPrdFrame[0]}
  [971] = {x=-26.59, y=15.422, z=13.967, rx=-179.103, ry=-1.546, rz=135.193, fatherId=fPrdFrame[0]}
  [972] = {x=-27.259, y=14.224, z=13.967, rx=-179.181, ry=-1.589, rz=135.192, fatherId=fPrdFrame[0]}
  [973] = {x=-28.105, y=12.495, z=13.968, rx=-179.273, ry=-1.634, rz=135.191, fatherId=fPrdFrame[0]}
  [974] = {x=-28.838, y=10.717, z=13.968, rx=-179.377, ry=-1.677, rz=135.19, fatherId=fPrdFrame[0]}
  [975] = {x=-29.365, y=9.197, z=13.968, rx=-179.465, ry=-1.708, rz=135.189, fatherId=fPrdFrame[0]}
  [976] = {x=-29.889, y=7.347, z=13.968, rx=-179.573, ry=-1.738, rz=135.187, fatherId=fPrdFrame[0]}
  [977] = {x=-30.295, y=5.468, z=13.969, rx=-179.682, ry=-1.762, rz=135.186, fatherId=fPrdFrame[0]}
  [978] = {x=-30.544, y=3.874, z=13.969, rx=-179.775, ry=-1.776, rz=135.184, fatherId=fPrdFrame[0]}
  [979] = {x=-30.732, y=1.961, z=13.969, rx=-179.886, ry=-1.787, rz=135.183, fatherId=fPrdFrame[0]}
  [980] = {x=-30.8, y=0.04, z=13.969, rx=-179.998, ry=-1.791, rz=135.181, fatherId=fPrdFrame[0]}
  [981] = {x=-30.765, y=-1.589, z=13.969, rx=179.913, ry=-1.789, rz=135.179, fatherId=fPrdFrame[0]}
  [982] = {x=-30.667, y=-2.969, z=13.969, rx=179.827, ry=-1.782, rz=135.178, fatherId=fPrdFrame[0]}
  [983] = {x=-30.507, y=-4.346, z=13.97, rx=179.747, ry=-1.773, rz=135.177, fatherId=fPrdFrame[0]}
  [984] = {x=-30.286, y=-5.712, z=13.97, rx=179.662, ry=-1.759, rz=135.176, fatherId=fPrdFrame[0]}
  [985] = {x=-29.877, y=-7.592, z=13.97, rx=179.559, ry=-1.736, rz=135.174, fatherId=fPrdFrame[0]}
  [986] = {x=-29.355, y=-9.442, z=13.97, rx=179.451, ry=-1.706, rz=135.173, fatherId=fPrdFrame[0]}
  [987] = {x=-28.721, y=-11.258, z=13.97, rx=179.346, ry=-1.669, rz=135.171, fatherId=fPrdFrame[0]}
  [988] = {x=-27.978, y=-13.031, z=13.971, rx=179.243, ry=-1.626, rz=135.17, fatherId=fPrdFrame[0]}
  [989] = {x=-27.129, y=-14.756, z=13.971, rx=179.143, ry=-1.576, rz=135.169, fatherId=fPrdFrame[0]}
  [990] = {x=-26.175, y=-16.425, z=13.972, rx=179.046, ry=-1.52, rz=135.168, fatherId=fPrdFrame[0]}
  [991] = {x=-25.119, y=-18.032, z=13.972, rx=178.952, ry=-1.459, rz=135.167, fatherId=fPrdFrame[0]}
  [992] = {x=-24.163, y=-19.321, z=13.973, rx=178.878, ry=-1.403, rz=135.167, fatherId=fPrdFrame[0]}
  [993] = {x=-23.325, y=-20.344, z=13.973, rx=178.817, ry=-1.354, rz=135.167, fatherId=fPrdFrame[0]}
  [994] = {x=-22.031, y=-21.767, z=13.974, rx=178.735, ry=-1.28, rz=135.167, fatherId=fPrdFrame[0]}
  [995] = {x=-20.651, y=-23.106, z=13.974, rx=178.658, ry=-1.2, rz=135.167, fatherId=fPrdFrame[0]}
  [996] = {x=-19.192, y=-24.358, z=13.975, rx=178.586, ry=-1.115, rz=135.167, fatherId=fPrdFrame[0]}
  [997] = {x=-17.641, y=-25.496, z=13.975, rx=178.431, ry=-1.093, rz=135.166, fatherId=fPrdFrame[0]}
  [998] = {x=-16.044, y=-26.564, z=13.976, rx=178.39, ry=-0.98, rz=135.167, fatherId=fPrdFrame[0]}
  [999] = {x=-14.384, y=-27.531, z=13.977, rx=178.348, ry=-0.869, rz=135.168, fatherId=fPrdFrame[0]}
string sFileName = "Disk://txt/TEST"
string sMoveMode[1000]
  [0] = "MOVEJ"
  [1] = "MOVEL"
  [2] = "MOVEL"
  [3] = "MOVEL"
  [4] = "MOVEL"
  [5] = "MOVEL"
  [6] = "MOVEL"
  [7] = "MOVEL"
  [8] = "MOVEL"
  [9] = "MOVEL"
  [10] = "MOVEL"
  [11] = "MOVEL"
  [12] = "MOVEL"
  [13] = "MOVEL"
  [14] = "MOVEL"
  [15] = "MOVEL"
  [16] = "MOVEL"
  [17] = "MOVEL"
  [18] = "MOVEL"
  [19] = "MOVEL"
  [20] = "MOVEL"
  [21] = "MOVEL"
  [22] = "MOVEL"
  [23] = "MOVEL"
  [24] = "MOVEL"
  [25] = "MOVEL"
  [26] = "MOVEL"
  [27] = "MOVEL"
  [28] = "MOVEL"
  [29] = "MOVEL"
  [30] = "MOVEL"
  [31] = "MOVEL"
  [32] = "MOVEL"
  [33] = "MOVEL"
  [34] = "MOVEL"
  [35] = "MOVEL"
  [36] = "MOVEL"
  [37] = "MOVEL"
  [38] = "MOVEL"
  [39] = "MOVEL"
  [40] = "MOVEL"
  [41] = "MOVEL"
  [42] = "MOVEL"
  [43] = "MOVEL"
  [44] = "MOVEL"
  [45] = "MOVEL"
  [46] = "MOVEL"
  [47] = "MOVEL"
  [48] = "MOVEL"
  [49] = "MOVEL"
  [50] = "MOVEL"
  [51] = "MOVEL"
  [52] = "MOVEL"
  [53] = "MOVEL"
  [54] = "MOVEL"
  [55] = "MOVEL"
  [56] = "MOVEL"
  [57] = "MOVEL"
  [58] = "MOVEL"
  [59] = "MOVEL"
  [60] = "MOVEL"
  [61] = "MOVEL"
  [62] = "MOVEL"
  [63] = "MOVEL"
  [64] = "MOVEL"
  [65] = "MOVEL"
  [66] = "MOVEL"
  [67] = "MOVEL"
  [68] = "MOVEL"
  [69] = "MOVEL"
  [70] = "MOVEL"
  [71] = "MOVEL"
  [72] = "MOVEL"
  [73] = "MOVEL"
  [74] = "MOVEL"
  [75] = "MOVEL"
  [76] = "MOVEL"
  [77] = "MOVEL"
  [78] = "MOVEL"
  [79] = "MOVEL"
  [80] = "MOVEL"
  [81] = "MOVEL"
  [82] = "MOVEL"
  [83] = "MOVEL"
  [84] = "MOVEL"
  [85] = "MOVEL"
  [86] = "MOVEL"
  [87] = "MOVEL"
  [88] = "MOVEL"
  [89] = "MOVEL"
  [90] = "MOVEL"
  [91] = "MOVEL"
  [92] = "MOVEL"
  [93] = "MOVEL"
  [94] = "MOVEL"
  [95] = "MOVEL"
  [96] = "MOVEL"
  [97] = "MOVEL"
  [98] = "MOVEL"
  [99] = "MOVEL"
  [100] = "MOVEL"
  [101] = "MOVEL"
  [102] = "MOVEL"
  [103] = "MOVEL"
  [104] = "MOVEL"
  [105] = "MOVEL"
  [106] = "MOVEL"
  [107] = "MOVEL"
  [108] = "MOVEL"
  [109] = "MOVEL"
  [110] = "MOVEL"
  [111] = "MOVEL"
  [112] = "MOVEL"
  [113] = "MOVEL"
  [114] = "MOVEL"
  [115] = "MOVEL"
  [116] = "MOVEL"
  [117] = "MOVEL"
  [118] = "MOVEL"
  [119] = "MOVEL"
  [120] = "MOVEL"
  [121] = "MOVEL"
  [122] = "MOVEL"
  [123] = "MOVEL"
  [124] = "MOVEL"
  [125] = "MOVEL"
  [126] = "MOVEL"
  [127] = "MOVEL"
  [128] = "MOVEL"
  [129] = "MOVEL"
  [130] = "MOVEL"
  [131] = "MOVEL"
  [132] = "MOVEL"
  [133] = "MOVEL"
  [134] = "MOVEL"
  [135] = "MOVEL"
  [136] = "MOVEL"
  [137] = "MOVEL"
  [138] = "MOVEL"
  [139] = "MOVEL"
  [140] = "MOVEL"
  [141] = "MOVEL"
  [142] = "MOVEL"
  [143] = "MOVEL"
  [144] = "MOVEL"
  [145] = "MOVEL"
  [146] = "MOVEL"
  [147] = "MOVEL"
  [148] = "MOVEL"
  [149] = "MOVEL"
  [150] = "MOVEL"
  [151] = "MOVEL"
  [152] = "MOVEL"
  [153] = "MOVEL"
  [154] = "MOVEL"
  [155] = "MOVEL"
  [156] = "MOVEL"
  [157] = "MOVEL"
  [158] = "MOVEL"
  [159] = "MOVEL"
  [160] = "MOVEL"
  [161] = "MOVEL"
  [162] = "MOVEL"
  [163] = "MOVEL"
  [164] = "MOVEL"
  [165] = "MOVEL"
  [166] = "MOVEL"
  [167] = "MOVEL"
  [168] = "MOVEL"
  [169] = "MOVEL"
  [170] = "MOVEL"
  [171] = "MOVEL"
  [172] = "MOVEL"
  [173] = "MOVEL"
  [174] = "MOVEL"
  [175] = "MOVEL"
  [176] = "MOVEL"
  [177] = "MOVEL"
  [178] = "MOVEL"
  [179] = "MOVEL"
  [180] = "MOVEL"
  [181] = "MOVEL"
  [182] = "MOVEL"
  [183] = "MOVEL"
  [184] = "MOVEL"
  [185] = "MOVEL"
  [186] = "MOVEL"
  [187] = "MOVEL"
  [188] = "MOVEL"
  [189] = "MOVEL"
  [190] = "MOVEL"
  [191] = "MOVEL"
  [192] = "MOVEL"
  [193] = "MOVEL"
  [194] = "MOVEL"
  [195] = "MOVEL"
  [196] = "MOVEL"
  [197] = "MOVEL"
  [198] = "MOVEL"
  [199] = "MOVEL"
  [200] = "MOVEL"
  [201] = "MOVEL"
  [202] = "MOVEL"
  [203] = "MOVEL"
  [204] = "MOVEL"
  [205] = "MOVEL"
  [206] = "MOVEL"
  [207] = "MOVEL"
  [208] = "MOVEL"
  [209] = "MOVEL"
  [210] = "MOVEL"
  [211] = "MOVEL"
  [212] = "MOVEL"
  [213] = "MOVEL"
  [214] = "MOVEL"
  [215] = "MOVEL"
  [216] = "MOVEL"
  [217] = "MOVEL"
  [218] = "MOVEL"
  [219] = "MOVEL"
  [220] = "MOVEL"
  [221] = "MOVEL"
  [222] = "MOVEL"
  [223] = "MOVEL"
  [224] = "MOVEL"
  [225] = "MOVEL"
  [226] = "MOVEL"
  [227] = "MOVEL"
  [228] = "MOVEL"
  [229] = "MOVEL"
  [230] = "MOVEL"
  [231] = "MOVEL"
  [232] = "MOVEL"
  [233] = "MOVEL"
  [234] = "MOVEL"
  [235] = "MOVEL"
  [236] = "MOVEL"
  [237] = "MOVEL"
  [238] = "MOVEL"
  [239] = "MOVEL"
  [240] = "MOVEL"
  [241] = "MOVEL"
  [242] = "MOVEL"
  [243] = "MOVEL"
  [244] = "MOVEL"
  [245] = "MOVEL"
  [246] = "MOVEL"
  [247] = "MOVEL"
  [248] = "MOVEL"
  [249] = "MOVEL"
  [250] = "MOVEL"
  [251] = "MOVEL"
  [252] = "MOVEL"
  [253] = "MOVEL"
  [254] = "MOVEL"
  [255] = "MOVEL"
  [256] = "MOVEL"
  [257] = "MOVEL"
  [258] = "MOVEL"
  [259] = "MOVEL"
  [260] = "MOVEL"
  [261] = "MOVEL"
  [262] = "MOVEL"
  [263] = "MOVEL"
  [264] = "MOVEL"
  [265] = "MOVEL"
  [266] = "MOVEL"
  [267] = "MOVEL"
  [268] = "MOVEL"
  [269] = "MOVEL"
  [270] = "MOVEL"
  [271] = "MOVEL"
  [272] = "MOVEL"
  [273] = "MOVEL"
  [274] = "MOVEL"
  [275] = "MOVEL"
  [276] = "MOVEL"
  [277] = "MOVEL"
  [278] = "MOVEL"
  [279] = "MOVEL"
  [280] = "MOVEL"
  [281] = "MOVEL"
  [282] = "MOVEL"
  [283] = "MOVEL"
  [284] = "MOVEL"
  [285] = "MOVEL"
  [286] = "MOVEL"
  [287] = "MOVEL"
  [288] = "MOVEL"
  [289] = "MOVEL"
  [290] = "MOVEL"
  [291] = "MOVEL"
  [292] = "MOVEL"
  [293] = "MOVEL"
  [294] = "MOVEL"
  [295] = "MOVEL"
  [296] = "MOVEL"
  [297] = "MOVEL"
  [298] = "MOVEL"
  [299] = "MOVEL"
  [300] = "MOVEL"
  [301] = "MOVEL"
  [302] = "MOVEL"
  [303] = "MOVEL"
  [304] = "MOVEL"
  [305] = "MOVEL"
  [306] = "MOVEL"
  [307] = "MOVEL"
  [308] = "MOVEL"
  [309] = "MOVEL"
  [310] = "MOVEL"
  [311] = "MOVEL"
  [312] = "MOVEL"
  [313] = "MOVEL"
  [314] = "MOVEL"
  [315] = "MOVEL"
  [316] = "MOVEL"
  [317] = "MOVEL"
  [318] = "MOVEL"
  [319] = "MOVEL"
  [320] = "MOVEL"
  [321] = "MOVEL"
  [322] = "MOVEL"
  [323] = "MOVEL"
  [324] = "MOVEL"
  [325] = "MOVEL"
  [326] = "MOVEL"
  [327] = "MOVEL"
  [328] = "MOVEL"
  [329] = "MOVEL"
  [330] = "MOVEL"
  [331] = "MOVEL"
  [332] = "MOVEL"
  [333] = "MOVEL"
  [334] = "MOVEL"
  [335] = "MOVEL"
  [336] = "MOVEL"
  [337] = "MOVEL"
  [338] = "MOVEL"
  [339] = "MOVEL"
  [340] = "MOVEL"
  [341] = "MOVEL"
  [342] = "MOVEL"
  [343] = "MOVEL"
  [344] = "MOVEL"
  [345] = "MOVEL"
  [346] = "MOVEL"
  [347] = "MOVEL"
  [348] = "MOVEL"
  [349] = "MOVEL"
  [350] = "MOVEL"
  [351] = "MOVEL"
  [352] = "MOVEL"
  [353] = "MOVEL"
  [354] = "MOVEL"
  [355] = "MOVEL"
  [356] = "MOVEL"
  [357] = "MOVEL"
  [358] = "MOVEL"
  [359] = "MOVEL"
  [360] = "MOVEL"
  [361] = "MOVEL"
  [362] = "MOVEL"
  [363] = "MOVEL"
  [364] = "MOVEL"
  [365] = "MOVEL"
  [366] = "MOVEL"
  [367] = "MOVEL"
  [368] = "MOVEL"
  [369] = "MOVEL"
  [370] = "MOVEL"
  [371] = "MOVEL"
  [372] = "MOVEL"
  [373] = "MOVEL"
  [374] = "MOVEL"
  [375] = "MOVEL"
  [376] = "MOVEL"
  [377] = "MOVEL"
  [378] = "MOVEL"
  [379] = "MOVEL"
  [380] = "MOVEL"
  [381] = "MOVEL"
  [382] = "MOVEL"
  [383] = "MOVEL"
  [384] = "MOVEL"
  [385] = "MOVEL"
  [386] = "MOVEL"
  [387] = "MOVEL"
  [388] = "MOVEL"
  [389] = "MOVEL"
  [390] = "MOVEL"
  [391] = "MOVEL"
  [392] = "MOVEL"
  [393] = "MOVEL"
  [394] = "MOVEL"
  [395] = "MOVEL"
  [396] = "MOVEL"
  [397] = "MOVEL"
  [398] = "MOVEL"
  [399] = "MOVEL"
  [400] = "MOVEL"
  [401] = "MOVEL"
  [402] = "MOVEL"
  [403] = "MOVEL"
  [404] = "MOVEL"
  [405] = "MOVEL"
  [406] = "MOVEL"
  [407] = "MOVEL"
  [408] = "MOVEL"
  [409] = "MOVEL"
  [410] = "MOVEL"
  [411] = "MOVEL"
  [412] = "MOVEL"
  [413] = "MOVEL"
  [414] = "MOVEL"
  [415] = "MOVEL"
  [416] = "MOVEL"
  [417] = "MOVEL"
  [418] = "MOVEL"
  [419] = "MOVEL"
  [420] = "MOVEL"
  [421] = "MOVEL"
  [422] = "MOVEL"
  [423] = "MOVEL"
  [424] = "MOVEL"
  [425] = "MOVEL"
  [426] = "MOVEL"
  [427] = "MOVEL"
  [428] = "MOVEL"
  [429] = "MOVEL"
  [430] = "MOVEL"
  [431] = "MOVEL"
  [432] = "MOVEL"
  [433] = "MOVEL"
  [434] = "MOVEL"
  [435] = "MOVEL"
  [436] = "MOVEL"
  [437] = "MOVEL"
  [438] = "MOVEL"
  [439] = "MOVEL"
  [440] = "MOVEL"
  [441] = "MOVEL"
  [442] = "MOVEL"
  [443] = "MOVEL"
  [444] = "MOVEL"
  [445] = "MOVEL"
  [446] = "MOVEL"
  [447] = "MOVEL"
  [448] = "MOVEL"
  [449] = "MOVEL"
  [450] = "MOVEL"
  [451] = "MOVEL"
  [452] = "MOVEL"
  [453] = "MOVEL"
  [454] = "MOVEL"
  [455] = "MOVEL"
  [456] = "MOVEL"
  [457] = "MOVEL"
  [458] = "MOVEL"
  [459] = "MOVEL"
  [460] = "MOVEL"
  [461] = "MOVEL"
  [462] = "MOVEL"
  [463] = "MOVEL"
  [464] = "MOVEL"
  [465] = "MOVEL"
  [466] = "MOVEL"
  [467] = "MOVEL"
  [468] = "MOVEL"
  [469] = "MOVEL"
  [470] = "MOVEL"
  [471] = "MOVEL"
  [472] = "MOVEL"
  [473] = "MOVEL"
  [474] = "MOVEL"
  [475] = "MOVEL"
  [476] = "MOVEL"
  [477] = "MOVEL"
  [478] = "MOVEL"
  [479] = "MOVEL"
  [480] = "MOVEL"
  [481] = "MOVEL"
  [482] = "MOVEL"
  [483] = "MOVEL"
  [484] = "MOVEL"
  [485] = "MOVEL"
  [486] = "MOVEL"
  [487] = "MOVEL"
  [488] = "MOVEL"
  [489] = "MOVEL"
  [490] = "MOVEL"
  [491] = "MOVEL"
  [492] = "MOVEL"
  [493] = "MOVEL"
  [494] = "MOVEL"
  [495] = "MOVEL"
  [496] = "MOVEL"
  [497] = "MOVEL"
  [498] = "MOVEL"
  [499] = "MOVEL"
  [500] = "MOVEL"
  [501] = "MOVEL"
  [502] = "MOVEL"
  [503] = "MOVEL"
  [504] = "MOVEL"
  [505] = "MOVEL"
  [506] = "MOVEL"
  [507] = "MOVEL"
  [508] = "MOVEL"
  [509] = "MOVEL"
  [510] = "MOVEL"
  [511] = "MOVEL"
  [512] = "MOVEL"
  [513] = "MOVEL"
  [514] = "MOVEL"
  [515] = "MOVEL"
  [516] = "MOVEL"
  [517] = "MOVEL"
  [518] = "MOVEL"
  [519] = "MOVEL"
  [520] = "MOVEL"
  [521] = "MOVEL"
  [522] = "MOVEL"
  [523] = "MOVEL"
  [524] = "MOVEL"
  [525] = "MOVEL"
  [526] = "MOVEL"
  [527] = "MOVEL"
  [528] = "MOVEL"
  [529] = "MOVEL"
  [530] = "MOVEL"
  [531] = "MOVEL"
  [532] = "MOVEL"
  [533] = "MOVEL"
  [534] = "MOVEL"
  [535] = "MOVEL"
  [536] = "MOVEL"
  [537] = "MOVEL"
  [538] = "MOVEL"
  [539] = "MOVEL"
  [540] = "MOVEL"
  [541] = "MOVEL"
  [542] = "MOVEL"
  [543] = "MOVEL"
  [544] = "MOVEL"
  [545] = "MOVEL"
  [546] = "MOVEL"
  [547] = "MOVEL"
  [548] = "MOVEL"
  [549] = "MOVEL"
  [550] = "MOVEL"
  [551] = "MOVEL"
  [552] = "MOVEL"
  [553] = "MOVEL"
  [554] = "MOVEL"
  [555] = "MOVEL"
  [556] = "MOVEL"
  [557] = "MOVEL"
  [558] = "MOVEL"
  [559] = "MOVEL"
  [560] = "MOVEL"
  [561] = "MOVEL"
  [562] = "MOVEL"
  [563] = "MOVEL"
  [564] = "MOVEL"
  [565] = "MOVEL"
  [566] = "MOVEL"
  [567] = "MOVEL"
  [568] = "MOVEL"
  [569] = "MOVEL"
  [570] = "MOVEL"
  [571] = "MOVEL"
  [572] = "MOVEL"
  [573] = "MOVEL"
  [574] = "MOVEL"
  [575] = "MOVEL"
  [576] = "MOVEL"
  [577] = "MOVEL"
  [578] = "MOVEL"
  [579] = "MOVEL"
  [580] = "MOVEL"
  [581] = "MOVEL"
  [582] = "MOVEL"
  [583] = "MOVEL"
  [584] = "MOVEL"
  [585] = "MOVEL"
  [586] = "MOVEL"
  [587] = "MOVEL"
  [588] = "MOVEL"
  [589] = "MOVEL"
  [590] = "MOVEL"
  [591] = "MOVEL"
  [592] = "MOVEL"
  [593] = "MOVEL"
  [594] = "MOVEL"
  [595] = "MOVEL"
  [596] = "MOVEL"
  [597] = "MOVEL"
  [598] = "MOVEL"
  [599] = "MOVEL"
  [600] = "MOVEL"
  [601] = "MOVEL"
  [602] = "MOVEL"
  [603] = "MOVEL"
  [604] = "MOVEL"
  [605] = "MOVEL"
  [606] = "MOVEL"
  [607] = "MOVEL"
  [608] = "MOVEL"
  [609] = "MOVEL"
  [610] = "MOVEL"
  [611] = "MOVEL"
  [612] = "MOVEL"
  [613] = "MOVEL"
  [614] = "MOVEL"
  [615] = "MOVEL"
  [616] = "MOVEL"
  [617] = "MOVEL"
  [618] = "MOVEL"
  [619] = "MOVEL"
  [620] = "MOVEL"
  [621] = "MOVEL"
  [622] = "MOVEL"
  [623] = "MOVEL"
  [624] = "MOVEL"
  [625] = "MOVEL"
  [626] = "MOVEL"
  [627] = "MOVEL"
  [628] = "MOVEL"
  [629] = "MOVEL"
  [630] = "MOVEL"
  [631] = "MOVEL"
  [632] = "MOVEL"
  [633] = "MOVEL"
  [634] = "MOVEL"
  [635] = "MOVEL"
  [636] = "MOVEL"
  [637] = "MOVEL"
  [638] = "MOVEL"
  [639] = "MOVEL"
  [640] = "MOVEL"
  [641] = "MOVEL"
  [642] = "MOVEL"
  [643] = "MOVEL"
  [644] = "MOVEL"
  [645] = "MOVEL"
  [646] = "MOVEL"
  [647] = "MOVEL"
  [648] = "MOVEL"
  [649] = "MOVEL"
  [650] = "MOVEL"
  [651] = "MOVEL"
  [652] = "MOVEL"
  [653] = "MOVEL"
  [654] = "MOVEL"
  [655] = "MOVEL"
  [656] = "MOVEL"
  [657] = "MOVEL"
  [658] = "MOVEL"
  [659] = "MOVEL"
  [660] = "MOVEL"
  [661] = "MOVEL"
  [662] = "MOVEL"
  [663] = "MOVEL"
  [664] = "MOVEL"
  [665] = "MOVEL"
  [666] = "MOVEL"
  [667] = "MOVEL"
  [668] = "MOVEL"
  [669] = "MOVEL"
  [670] = "MOVEL"
  [671] = "MOVEL"
  [672] = "MOVEL"
  [673] = "MOVEL"
  [674] = "MOVEL"
  [675] = "MOVEL"
  [676] = "MOVEL"
  [677] = "MOVEL"
  [678] = "MOVEL"
  [679] = "MOVEL"
  [680] = "MOVEL"
  [681] = "MOVEL"
  [682] = "MOVEL"
  [683] = "MOVEL"
  [684] = "MOVEL"
  [685] = "MOVEL"
  [686] = "MOVEL"
  [687] = "MOVEL"
  [688] = "MOVEL"
  [689] = "MOVEL"
  [690] = "MOVEL"
  [691] = "MOVEL"
  [692] = "MOVEL"
  [693] = "MOVEL"
  [694] = "MOVEL"
  [695] = "MOVEL"
  [696] = "MOVEL"
  [697] = "MOVEL"
  [698] = "MOVEL"
  [699] = "MOVEL"
  [700] = "MOVEL"
  [701] = "MOVEL"
  [702] = "MOVEL"
  [703] = "MOVEL"
  [704] = "MOVEL"
  [705] = "MOVEL"
  [706] = "MOVEL"
  [707] = "MOVEL"
  [708] = "MOVEL"
  [709] = "MOVEL"
  [710] = "MOVEL"
  [711] = "MOVEL"
  [712] = "MOVEL"
  [713] = "MOVEL"
  [714] = "MOVEL"
  [715] = "MOVEL"
  [716] = "MOVEL"
  [717] = "MOVEL"
  [718] = "MOVEL"
  [719] = "MOVEL"
  [720] = "MOVEL"
  [721] = "MOVEL"
  [722] = "MOVEL"
  [723] = "MOVEL"
  [724] = "MOVEL"
  [725] = "MOVEL"
  [726] = "MOVEL"
  [727] = "MOVEL"
  [728] = "MOVEL"
  [729] = "MOVEL"
  [730] = "MOVEL"
  [731] = "MOVEL"
  [732] = "MOVEL"
  [733] = "MOVEL"
  [734] = "MOVEL"
  [735] = "MOVEL"
  [736] = "MOVEL"
  [737] = "MOVEL"
  [738] = "MOVEL"
  [739] = "MOVEL"
  [740] = "MOVEL"
  [741] = "MOVEL"
  [742] = "MOVEL"
  [743] = "MOVEL"
  [744] = "MOVEL"
  [745] = "MOVEL"
  [746] = "MOVEL"
  [747] = "MOVEL"
  [748] = "MOVEL"
  [749] = "MOVEL"
  [750] = "MOVEL"
  [751] = "MOVEL"
  [752] = "MOVEL"
  [753] = "MOVEL"
  [754] = "MOVEL"
  [755] = "MOVEL"
  [756] = "MOVEL"
  [757] = "MOVEL"
  [758] = "MOVEL"
  [759] = "MOVEL"
  [760] = "MOVEL"
  [761] = "MOVEL"
  [762] = "MOVEL"
  [763] = "MOVEL"
  [764] = "MOVEL"
  [765] = "MOVEL"
  [766] = "MOVEL"
  [767] = "MOVEL"
  [768] = "MOVEL"
  [769] = "MOVEL"
  [770] = "MOVEL"
  [771] = "MOVEL"
  [772] = "MOVEL"
  [773] = "MOVEL"
  [774] = "MOVEL"
  [775] = "MOVEL"
  [776] = "MOVEL"
  [777] = "MOVEL"
  [778] = "MOVEL"
  [779] = "MOVEL"
  [780] = "MOVEL"
  [781] = "MOVEL"
  [782] = "MOVEL"
  [783] = "MOVEL"
  [784] = "MOVEL"
  [785] = "MOVEL"
  [786] = "MOVEL"
  [787] = "MOVEL"
  [788] = "MOVEL"
  [789] = "MOVEL"
  [790] = "MOVEL"
  [791] = "MOVEL"
  [792] = "MOVEL"
  [793] = "MOVEL"
  [794] = "MOVEL"
  [795] = "MOVEL"
  [796] = "MOVEL"
  [797] = "MOVEL"
  [798] = "MOVEL"
  [799] = "MOVEL"
  [800] = "MOVEL"
  [801] = "MOVEL"
  [802] = "MOVEL"
  [803] = "MOVEL"
  [804] = "MOVEL"
  [805] = "MOVEL"
  [806] = "MOVEL"
  [807] = "MOVEL"
  [808] = "MOVEL"
  [809] = "MOVEL"
  [810] = "MOVEL"
  [811] = "MOVEL"
  [812] = "MOVEL"
  [813] = "MOVEL"
  [814] = "MOVEL"
  [815] = "MOVEL"
  [816] = "MOVEL"
  [817] = "MOVEL"
  [818] = "MOVEL"
  [819] = "MOVEL"
  [820] = "MOVEL"
  [821] = "MOVEL"
  [822] = "MOVEL"
  [823] = "MOVEL"
  [824] = "MOVEL"
  [825] = "MOVEL"
  [826] = "MOVEL"
  [827] = "MOVEL"
  [828] = "MOVEL"
  [829] = "MOVEL"
  [830] = "MOVEL"
  [831] = "MOVEL"
  [832] = "MOVEL"
  [833] = "MOVEL"
  [834] = "MOVEL"
  [835] = "MOVEL"
  [836] = "MOVEL"
  [837] = "MOVEL"
  [838] = "MOVEL"
  [839] = "MOVEL"
  [840] = "MOVEL"
  [841] = "MOVEL"
  [842] = "MOVEL"
  [843] = "MOVEL"
  [844] = "MOVEL"
  [845] = "MOVEL"
  [846] = "MOVEL"
  [847] = "MOVEL"
  [848] = "MOVEL"
  [849] = "MOVEL"
  [850] = "MOVEL"
  [851] = "MOVEL"
  [852] = "MOVEL"
  [853] = "MOVEL"
  [854] = "MOVEL"
  [855] = "MOVEL"
  [856] = "MOVEL"
  [857] = "MOVEL"
  [858] = "MOVEL"
  [859] = "MOVEL"
  [860] = "MOVEL"
  [861] = "MOVEL"
  [862] = "MOVEL"
  [863] = "MOVEL"
  [864] = "MOVEL"
  [865] = "MOVEL"
  [866] = "MOVEL"
  [867] = "MOVEL"
  [868] = "MOVEL"
  [869] = "MOVEL"
  [870] = "MOVEL"
  [871] = "MOVEL"
  [872] = "MOVEL"
  [873] = "MOVEL"
  [874] = "MOVEL"
  [875] = "MOVEL"
  [876] = "MOVEL"
  [877] = "MOVEL"
  [878] = "MOVEL"
  [879] = "MOVEL"
  [880] = "MOVEL"
  [881] = "MOVEL"
  [882] = "MOVEL"
  [883] = "MOVEL"
  [884] = "MOVEL"
  [885] = "MOVEL"
  [886] = "MOVEL"
  [887] = "MOVEL"
  [888] = "MOVEL"
  [889] = "MOVEL"
  [890] = "MOVEL"
  [891] = "MOVEL"
  [892] = "MOVEL"
  [893] = "MOVEL"
  [894] = "MOVEL"
  [895] = "MOVEL"
  [896] = "MOVEL"
  [897] = "MOVEL"
  [898] = "MOVEL"
  [899] = "MOVEL"
  [900] = "MOVEL"
  [901] = "MOVEL"
  [902] = "MOVEL"
  [903] = "MOVEL"
  [904] = "MOVEL"
  [905] = "MOVEL"
  [906] = "MOVEL"
  [907] = "MOVEL"
  [908] = "MOVEL"
  [909] = "MOVEL"
  [910] = "MOVEL"
  [911] = "MOVEL"
  [912] = "MOVEL"
  [913] = "MOVEL"
  [914] = "MOVEL"
  [915] = "MOVEL"
  [916] = "MOVEL"
  [917] = "MOVEL"
  [918] = "MOVEL"
  [919] = "MOVEL"
  [920] = "MOVEL"
  [921] = "MOVEL"
  [922] = "MOVEL"
  [923] = "MOVEL"
  [924] = "MOVEL"
  [925] = "MOVEL"
  [926] = "MOVEL"
  [927] = "MOVEL"
  [928] = "MOVEL"
  [929] = "MOVEL"
  [930] = "MOVEL"
  [931] = "MOVEL"
  [932] = "MOVEL"
  [933] = "MOVEL"
  [934] = "MOVEL"
  [935] = "MOVEL"
  [936] = "MOVEL"
  [937] = "MOVEL"
  [938] = "MOVEL"
  [939] = "MOVEL"
  [940] = "MOVEL"
  [941] = "MOVEL"
  [942] = "MOVEL"
  [943] = "MOVEL"
  [944] = "MOVEL"
  [945] = "MOVEL"
  [946] = "MOVEL"
  [947] = "MOVEL"
  [948] = "MOVEL"
  [949] = "MOVEL"
  [950] = "MOVEL"
  [951] = "MOVEL"
  [952] = "MOVEL"
  [953] = "MOVEL"
  [954] = "MOVEL"
  [955] = "MOVEL"
  [956] = "MOVEL"
  [957] = "MOVEL"
  [958] = "MOVEL"
  [959] = "MOVEL"
  [960] = "MOVEL"
  [961] = "MOVEL"
  [962] = "MOVEL"
  [963] = "MOVEL"
  [964] = "MOVEL"
  [965] = "MOVEL"
  [966] = "MOVEL"
  [967] = "MOVEL"
  [968] = "MOVEL"
  [969] = "MOVEL"
  [970] = "MOVEL"
  [971] = "MOVEL"
  [972] = "MOVEL"
  [973] = "MOVEL"
  [974] = "MOVEL"
  [975] = "MOVEL"
  [976] = "MOVEL"
  [977] = "MOVEL"
  [978] = "MOVEL"
  [979] = "MOVEL"
  [980] = "MOVEL"
  [981] = "MOVEL"
  [982] = "MOVEL"
  [983] = "MOVEL"
  [984] = "MOVEL"
  [985] = "MOVEL"
  [986] = "MOVEL"
  [987] = "MOVEL"
  [988] = "MOVEL"
  [989] = "MOVEL"
  [990] = "MOVEL"
  [991] = "MOVEL"
  [992] = "MOVEL"
  [993] = "MOVEL"
  [994] = "MOVEL"
  [995] = "MOVEL"
  [996] = "MOVEL"
  [997] = "MOVEL"
  [998] = "MOVEL"
  [999] = "MOVEL"
string sPrdID = "TEST"
string sSpeedDate = "  5.4 "
public tool tPrdTool = {fatherId=flange[0], ioLink=valve1}
trsf trPrdFrmOffset

--- start.pgx ---
program start()
begin
  if taskStatus("trajManage")!=-1
    taskKill("trajManage")
    wait(taskStatus("trajManage")==-1)
  endIf
  if taskStatus("motion")!=-1
    taskKill("motion")
    wait(taskStatus("motion")==-1)
  endIf
  bCycleEnd=false
  bCycle=true
  bResumeCycle=true
  taskCreate "trajManage",95,fileRead("test.txt")
  taskCreate "motion",98,trajGrind()

end

--- fileRead.pgx ---
public program fileRead(string x_sTxtName)
  local bool l_bReadHead
  local num l_nRead
  local string l_sRead
  local string l_sSign[2]
  local string l_sDate[2]
  local num i
begin
  call init()
  bCycle=true
  //打开文件
  sFileName="Disk://txt/"+x_sTxtName
  if $fileExists(sFileName)==false
    popUpMsg(sFileName+"文件不存在")
    bCycle=false
    bCycleEnd=true
    bResumeCycle=false
    return
  endIf


  //读取文件头
  nFileId=$fileOpen(sFileName,"r")
  call ReadHead(nFileId,l_bReadHead,sPrdID,tPrdTool,jPrdHome,fPrdFrame,trPrdFrmOffset,nTotalTrajs)
  $fileClose(nFileId)
  //判断头文件是否正确
  if l_bReadHead==false
    popUpMsg("头文件格式或内容错误")
    return
  endIf
  //关键数据核对检查
  // libSave()






  bTxtHeadOk=true
  l_sSign[0]=""
  l_sSign[1]=""
  //
  nFileId=$fileOpen(sFileName,"r")
  //文件内容读取
  //从"BYPASS=FALSE"标示符开始采集数据
  do
    l_nRead=$fileGet(nFileId,l_sRead,1)
    call getStrSign(l_sRead,l_sSign)
    //路径结束标志
    if l_sSign[1]=="END"
      if nCurrentTraj<nTotalTrajs
        nCurrentTraj=nCurrentTraj+1
      endIf
    endIf
  until l_sSign[0]=="BYPASS" and l_sSign[1]=="FALSE"
  bBYPASS=false
  do
    //等待读取信息
    while (nReadPtr+nThousandRead*1000+900<nThousandWrite*1000+nWritePtr or nReadJnt+nHundredRead*100+50<nWriteJnt+nHundredWrite*100) and !bResumeCycle
      delay(0)
    endWhile
    l_nRead=$fileGet(nFileId,l_sRead,1)
    call getStrSign(l_sRead,l_sSign)
    //路径是否过滤
    if l_sSign=="BYPASS" and l_sSign[1]=="TRUE"
      bBYPASS=true
    endIf
    if l_sSign=="BYPASS" and l_sSign[1]=="FALSE"
      bBYPASS=false
    endIf
    if !bBYPASS
      //获取是否从TXT获得速度信息
//      if !bGetSpeed
//        if l_sSign=="GETSPEED" and l_sSign[1]=="TRUE"
//          bGetSpeed=true
//          date:libSave()
//        endIf
//      endIf
      //获取转台信息,判断模式
      if date:bWorTbMoving==false
        if l_sSign=="WORKTABLEMODE" and l_sSign[1]=="TRUE"
          date:bWorTbMoving=true
          //2015.06.23
          //date:libSave()
        endIf
      endIf
      //MOVEJ情形
      if l_sSign=="MOVEJ"
        call getStrDate(l_sSign[1],l_sDate)
        sMoveMode[nWritePtr]="MOVEJ"
        call getJointDate(l_sDate[0],jJointRead[nWriteJnt])
        //2015.02.05
        call getSpeedDate(l_sDate[1],mSpdOfJnt[nWriteJnt])
        nWriteJnt=nWriteJnt+1
        if nWriteJnt>99
          nWriteJnt=0
          nHundredWrite=nHundredWrite+1
        endIf
        nWritePtr=nWritePtr+1
        if nWritePtr>999
          nWritePtr=0
          nThousandWrite=nThousandWrite+1
        endIf
      endIf
      //MOVEL情形
      if l_sSign=="MOVEL"
        call getStrDate(l_sSign[1],l_sDate)
        sMoveMode[nWritePtr]="MOVEL"
        link(pPointRead[nWritePtr],fPrdFrame)
        call getPointDate(l_sDate[0],pPointRead[nWritePtr])
        //从TXT中获得机器人速度参数
        if bGetSpeed
          call getSpeedDate(l_sDate[1],mSpdOfPt[nWritePtr])
        endIf
        //          //转台转动情形
        //          if date:bWorTbMoving==true
        //            nDistToOrign=sqrt(pPointRead[nWritePtr].trsf.x*pPointRead[nWritePtr].trsf.x+pPointRead[nWritePtr].trsf.y*pPointRead[nWritePtr].trsf.y)
        //            //
        //            //修改机器人移动速度：速度关系式v=v(1-k*d/r)
        //            mSpdOfPt[nWritePtr].tvel=mSpdOfPt[nWritePtr].tvel*(1-0.5*nDistToOrign/nPrdRadius)
        //            //
        //          endIf
        nWritePtr=nWritePtr+1
        if nWritePtr>999
          nWritePtr=0
          nThousandWrite=nThousandWrite+1
        endIf
      endIf
    endIf
    //路径结束标志
    if l_sSign[1]=="END"
      if nCurrentTraj<nTotalTrajs
        if size(nPtOfTraj)<nCurrentTraj+1
          $dins(nPtOfTraj,size(nPtOfTraj)-1)
        endIf
        nPtOfTraj[nCurrentTraj]=nThousandWrite*1000+nWritePtr
        nCurrentTraj=nCurrentTraj+1
        l_sSign[1]=""
      endIf
    endIf
    delay(0)
  until nCurrentTraj==nTotalTrajs
  bWriteEnd=true
  $fileClose(nFileId)


  //libSave()
end

--- NCVetor.pgx ---
program NCVetor(trsf x_trFrame, trsf& x_trNC)
  local trsf l_trTrsf
begin


//  x_trFrame.x=x_trFrame.y=x_trFrame.z=0
//
//  //l_trTrsf=x_trFrame*{0,0,0,180,0,180}*{0,0,0,x_trNC.rx,x_trNC.ry,x_trNC.rz}
//  //l_trTrsf=!x_trFrame*l_trTrsf
//
//  l_trTrsf={0,0,0,180,0,180}*{0,0,0,x_trNC.rx,x_trNC.ry,x_trNC.rz}




//  x_trNC.rx=l_trTrsf.rx
//  x_trNC.ry=l_trTrsf.ry
//  x_trNC.rz=l_trTrsf.rz


end

--- ReadHead.pgx ---
program ReadHead(num x_nFileID, bool& x_bHeaderOk, string& x_sPrdID, tool& x_tTool, joint& x_jHome, frame& x_fFrame, trsf& x_trOffset, num& x_nTotalTrajs)
  local num l_nRead
  local string l_sRead
  local num l_nFind
  local string l_sSplit[2]
  local string l_sValue[6]
  local bool b[7]
begin
  if nFileId>=0 or nFileId<=9
    x_bHeaderOk=false
    bMatlab=false
    while !x_bHeaderOk
      l_nRead=$fileGet(nFileId,l_sRead,1)
      //
      call split(l_sRead,"=",l_sSplit)
      call split(l_sSplit[1],",",l_sValue)
      //
      switch l_sSplit[0]
        case "PRODUCTID"
          x_sPrdID=l_sValue[0]
        break
        case "TOOL"
          l_sValue[0]=toNum(l_sValue[0],x_tTool.trsf.x,b[1])
          l_sValue[1]=toNum(l_sValue[1],x_tTool.trsf.y,b[2])
          l_sValue[2]=toNum(l_sValue[2],x_tTool.trsf.z,b[3])
          l_sValue[3]=toNum(l_sValue[3],x_tTool.trsf.rx,b[4])
          l_sValue[4]=toNum(l_sValue[4],x_tTool.trsf.ry,b[5])
          l_sValue[5]=toNum(l_sValue[5],x_tTool.trsf.rz,b[6])
        break
        case "HOME"
          l_sValue[0]=toNum(l_sValue[0],x_jHome.j1,b[1])
          l_sValue[1]=toNum(l_sValue[1],x_jHome.j2,b[2])
          l_sValue[2]=toNum(l_sValue[2],x_jHome.j3,b[3])
          l_sValue[3]=toNum(l_sValue[3],x_jHome.j4,b[4])
          l_sValue[4]=toNum(l_sValue[4],x_jHome.j5,b[5])
          l_sValue[5]=toNum(l_sValue[5],x_jHome.j6,b[6])
        break
        case "FRAME"
          l_sValue[0]=toNum(l_sValue[0],x_fFrame.trsf.x,b[1])
          l_sValue[1]=toNum(l_sValue[1],x_fFrame.trsf.y,b[2])
          l_sValue[2]=toNum(l_sValue[2],x_fFrame.trsf.z,b[3])
          l_sValue[3]=toNum(l_sValue[3],x_fFrame.trsf.rx,b[4])
          l_sValue[4]=toNum(l_sValue[4],x_fFrame.trsf.ry,b[5])
          l_sValue[5]=toNum(l_sValue[5],x_fFrame.trsf.rz,b[6])
        break
        case "OFFSET"
          l_sValue[0]=toNum(l_sValue[0],x_trOffset.x,b[1])
          l_sValue[1]=toNum(l_sValue[1],x_trOffset.y,b[2])
          l_sValue[2]=toNum(l_sValue[2],x_trOffset.z,b[3])
          l_sValue[3]=toNum(l_sValue[3],x_trOffset.rx,b[4])
          l_sValue[4]=toNum(l_sValue[4],x_trOffset.ry,b[5])
          l_sValue[5]=toNum(l_sValue[5],x_trOffset.rz,b[6])
        break
        case "TOTALTRAJS"
          l_sValue[0]=toNum(l_sValue[0],x_nTotalTrajs,b[1])
        break

        case "OFFLINE"
//          bMatlab=true
//          x_fFrame.trsf={0,0,-13.488,0,0,0}*x_fFrame.trsf
        break

      endSwitch
      //当提取到=后面的"BEGIN"时,头文件读取结束
      if l_sSplit[1]=="BEGIN"
        x_bHeaderOk=true
      endIf
    endWhile
  else
    popUpMsg(sFileName+"does not open")
    logMsg(sFileName+"does not open")
    x_bHeaderOk=false
  endIf

end

--- Readme.pgx ---
program readme()
begin
  //Title :
  //
  //General description :
  //  This library is used to extract data from text file.
  //  It can also be used to meneage date and move the arm along resulting trajectory.
  //  There is a public program, named main()
  //
  //Hardware required :
  //  - Robot system    : any 6 axis Staubli robot
  //  - Peripherals     : no peripherals required
  //
  //VAL3 options :
  //  - VAL3 version    : 7.3.1
  //  - VAL3 licenses   : no licenses required
  //  - VAL3 add-ons    : expansion (VAL3 add-ons are version specific in regards to the version of VAL3)
  //
  //Library version     : 7.3.1
  //
  //Public variables    : none
  //
  //Included libraries  : none
  //
  //Keywords            : tool, extraction, text files,
  //
end
